LIN {X 0,Y 456.406,Z 1058.133,A -85,B 0,C 180,E1 19306.793,E2 19306.793} C_VEL
LIN {X 0,Y 463.105,Z 1034.289,A -85,B 0,C 180,E1 19306.028,E2 19306.028} C_VEL
LIN {X 0,Y 471.257,Z 1002.523,A -85,B 0,C 180,E1 19305.397,E2 19305.397} C_VEL
LIN {X 0,Y 477.978,Z 976.833,A -85,B 0,C 180,E1 19305.03,E2 19305.03} C_VEL
LIN {X 0,Y 462.437,Z 1036.182,A -85,B 0,C 180,E1 19303.259,E2 19303.259} C_VEL
LIN {X 0,Y 455.558,Z 1059.774,A -85,B 0,C 180,E1 19302.278,E2 19302.278} C_VEL
LIN {X 0,Y 447.956,Z 1083.299,A -85,B 0,C 180,E1 19301.014,E2 19301.014} C_VEL
LIN {X 0,Y 440.173,Z 1105.866,A -85,B 0,C 180,E1 19299.498,E2 19299.498} C_VEL
LIN {X 0,Y 432.109,Z 1128.201,A -85,B 0,C 180,E1 19297.654,E2 19297.654} C_VEL
LIN {X 0,Y 424.459,Z 1148.843,A -85,B 0,C 180,E1 19295.581,E2 19295.581} C_VEL
LIN {X 0,Y 417.628,Z 1166.966,A -85,B 0,C 180,E1 19293.413,E2 19293.413} C_VEL
LIN {X 0,Y 410.886,Z 1184.567,A -85,B 0,C 180,E1 19290.895,E2 19290.895} C_VEL
LIN {X 0,Y 404.741,Z 1200.504,A -85,B 0,C 180,E1 19288.155,E2 19288.155} C_VEL
LIN {X 0,Y 399.298,Z 1214.717,A -85,B 0,C 180,E1 19285.195,E2 19285.195} C_VEL
LIN {X 0,Y 395.001,Z 1226.059,A -85,B 0,C 180,E1 19282.315,E2 19282.315} C_VEL
LIN {X 0,Y 391.557,Z 1235.554,A -85,B 0,C 180,E1 19279.389,E2 19279.389} C_VEL
LIN {X 0,Y 388.794,Z 1243.686,A -85,B 0,C 180,E1 19276.28,E2 19276.28} C_VEL
LIN {X 0,Y 386.823,Z 1250.051,A -85,B 0,C 180,E1 19273.148,E2 19273.148} C_VEL
LIN {X 0,Y 385.498,Z 1254.602,A -85,B 0,C 180,E1 19270.008,E2 19270.008} C_VEL
LIN {X 0,Y 384.741,Z 1257.556,A -85,B 0,C 180,E1 19266.866,E2 19266.866} C_VEL
LIN {X 0,Y 384.358,Z 1258.935,A -85,B 0,C 180,E1 19263.878,E2 19263.878} C_VEL
LIN {X 0,Y 384.196,Z 1258.702,A -85,B 0,C 180,E1 19260.895,E2 19260.895} C_VEL
LIN {X 0,Y 384.141,Z 1256.912,A -85,B 0,C 180,E1 19257.762,E2 19257.762} C_VEL
LIN {X 0,Y 384.207,Z 1253.678,A -85,B 0,C 180,E1 19254.774,E2 19254.774} C_VEL
LIN {X 0,Y 384.45,Z 1248.721,A -85,B 0,C 180,E1 19251.776,E2 19251.776} C_VEL
LIN {X 0,Y 385.024,Z 1241.729,A -85,B 0,C 180,E1 19248.617,E2 19248.617} C_VEL
LIN {X 0,Y 385.962,Z 1233.447,A -85,B 0,C 180,E1 19245.678,E2 19245.678} C_VEL
LIN {X 0,Y 387.402,Z 1223.201,A -85,B 0,C 180,E1 19242.733,E2 19242.733} C_VEL
LIN {X 0,Y 389.23,Z 1211.755,A -85,B 0,C 180,E1 19240.022,E2 19240.022} C_VEL
LIN {X 0,Y 391.588,Z 1198.234,A -85,B 0,C 180,E1 19237.321,E2 19237.321} C_VEL
LIN {X 0,Y 394.348,Z 1183.215,A -85,B 0,C 180,E1 19234.788,E2 19234.788} C_VEL
LIN {X 0,Y 397.336,Z 1167.26,A -85,B 0,C 180,E1 19232.498,E2 19232.498} C_VEL
LIN {X 0,Y 400.703,Z 1148.832,A -85,B 0,C 180,E1 19230.273,E2 19230.273} C_VEL
LIN {X 0,Y 404.024,Z 1129.942,A -85,B 0,C 180,E1 19228.354,E2 19228.354} C_VEL
LIN {X 0,Y 407.3,Z 1109.911,A -85,B 0,C 180,E1 19226.639,E2 19226.639} C_VEL
LIN {X 0,Y 410.601,Z 1088.057,A -85,B 0,C 180,E1 19225.091,E2 19225.091} C_VEL
LIN {X 0,Y 413.484,Z 1066.4,A -85,B 0,C 180,E1 19223.84,E2 19223.84} C_VEL
LIN {X 0,Y 416.065,Z 1043.427,A -85,B 0,C 180,E1 19222.783,E2 19222.783} C_VEL
LIN {X 0,Y 418.284,Z 1019.214,A -85,B 0,C 180,E1 19221.949,E2 19221.949} C_VEL
LIN {X 0,Y 420.646,Z 982.191,A -85,B 0,C 180,E1 19221.071,E2 19221.071} C_VEL
LIN {X 0,Y 434.104,Z 779.214,A -85,B 0,C 180,E1 19216.578,E2 19216.578} C_VEL
LIN {X 0,Y 417.769,Z 747.187,A -85,B 0,C 180,E1 19214.052,E2 19214.052} C_VEL
LIN {X 0,Y 402.103,Z 718.746,A -85,B 0,C 180,E1 19211.46,E2 19211.46} C_VEL
LIN {X 0,Y 397.559,Z 710.697,A -85,B 0,C 180,E1 19210.649,E2 19210.649} C_VEL
LIN {X 0,Y 389.693,Z 691.665,A -85,B 0,C 180,E1 19207.269,E2 19207.269} C_VEL
LIN {X 0,Y 386.803,Z 684.581,A -85,B 0,C 180,E1 19205.973,E2 19205.973} C_VEL
LIN {X 0,Y 386.779,Z 684.484,A -85,B 0,C 180,E1 19201.83,E2 19201.83} C_VEL
LIN {X 0,Y 386.786,Z 684.485,A -85,B 0,C 180,E1 19197.857,E2 19197.857} C_VEL
LIN {X 0,Y 386.792,Z 684.486,A -85,B 0,C 180,E1 19193.776,E2 19193.776} C_VEL
LIN {X 0,Y 386.789,Z 684.485,A -85,B 0,C 180,E1 19189.783,E2 19189.783} C_VEL
LIN {X 0,Y 386.784,Z 684.488,A -85,B 0,C 180,E1 19185.752,E2 19185.752} C_VEL
LIN {X 0,Y 386.779,Z 684.483,A -85,B 0,C 180,E1 19181.786,E2 19181.786} C_VEL
LIN {X 0,Y 386.794,Z 684.472,A -85,B 0,C 180,E1 19177.727,E2 19177.727} C_VEL
LIN {X 0,Y 386.778,Z 684.475,A -85,B 0,C 180,E1 19173.708,E2 19173.708} C_VEL
LIN {X 0,Y 386.78,Z 684.474,A -85,B 0,C 180,E1 19169.706,E2 19169.706} C_VEL
LIN {X 0,Y 386.785,Z 684.475,A -85,B 0,C 180,E1 19165.703,E2 19165.703} C_VEL
LIN {X 0,Y 386.786,Z 684.478,A -85,B 0,C 180,E1 19161.678,E2 19161.678} C_VEL
LIN {X 0,Y 386.788,Z 684.487,A -85,B 0,C 180,E1 19157.612,E2 19157.612} C_VEL
LIN {X 0,Y 386.781,Z 684.489,A -85,B 0,C 180,E1 19153.636,E2 19153.636} C_VEL
LIN {X 0,Y 386.781,Z 684.483,A -85,B 0,C 180,E1 19149.577,E2 19149.577} C_VEL
LIN {X 0,Y 386.797,Z 684.617,A -85,B 0,C 180,E1 19146.592,E2 19146.592} C_VEL
LIN {X 0,Y 388.136,Z 688.034,A -85,B 0,C 180,E1 19145.823,E2 19145.823} C_VEL
LIN {X 0,Y 392.774,Z 697.922,A -85,B 0,C 180,E1 19143.547,E2 19143.547} C_VEL
LIN {X 0,Y 399.276,Z 712.504,A -85,B 0,C 180,E1 19140.443,E2 19140.443} C_VEL
LIN {X 0,Y 406.573,Z 730.369,A -85,B 0,C 180,E1 19136.996,E2 19136.996} C_VEL
LIN {X 0,Y 413.648,Z 749.213,A -85,B 0,C 180,E1 19133.688,E2 19133.688} C_VEL
LIN {X 0,Y 420.237,Z 768.718,A -85,B 0,C 180,E1 19130.562,E2 19130.562} C_VEL
LIN {X 0,Y 423.081,Z 778.482,A -85,B 0,C 180,E1 19129.11,E2 19129.11} C_VEL
LIN {X 0,Y 422.399,Z 782.605,A -85,B 0,C 180,E1 19128.699,E2 19128.699} C_VEL
LIN {X 0,Y 420.547,Z 788.964,A -85,B 0,C 180,E1 19128.148,E2 19128.148} C_VEL
LIN {X 0,Y 412.54,Z 806.493,A -85,B 0,C 180,E1 19126.91,E2 19126.91} C_VEL
LIN {X 0,Y 411.039,Z 811.959,A -85,B 0,C 180,E1 19126.42,E2 19126.42} C_VEL
LIN {X 0,Y 404.701,Z 854.209,A -85,B 0,C 180,E1 19122.17,E2 19122.17} C_VEL
LIN {X 0,Y 398.898,Z 897.769,A -85,B 0,C 180,E1 19117.807,E2 19117.807} C_VEL
LIN {X 0,Y 396.431,Z 919.14,A -85,B 0,C 180,E1 19115.714,E2 19115.714} C_VEL
LIN {X 0,Y 396.961,Z 931.506,A -85,B 0,C 180,E1 19115.277,E2 19115.277} C_VEL
LIN {X 0,Y 391.461,Z 1014.878,A -85,B 0,C 180,E1 19112.751,E2 19112.751} C_VEL
LIN {X 0,Y 388.582,Z 1066.505,A -85,B 0,C 180,E1 19110.979,E2 19110.979} C_VEL
LIN {X 0,Y 387.682,Z 1083.198,A -85,B 0,C 180,E1 19110.195,E2 19110.195} C_VEL
LIN {X 0,Y 386.441,Z 1100.03,A -85,B 0,C 180,E1 19109.107,E2 19109.107} C_VEL
LIN {X 0,Y 385.089,Z 1114.976,A -85,B 0,C 180,E1 19107.864,E2 19107.864} C_VEL
LIN {X 0,Y 383.556,Z 1130.549,A -85,B 0,C 180,E1 19106.233,E2 19106.233} C_VEL
LIN {X 0,Y 382.067,Z 1144.335,A -85,B 0,C 180,E1 19104.425,E2 19104.425} C_VEL
LIN {X 0,Y 380.789,Z 1156.067,A -85,B 0,C 180,E1 19102.543,E2 19102.543} C_VEL
LIN {X 0,Y 379.604,Z 1167.141,A -85,B 0,C 180,E1 19100.337,E2 19100.337} C_VEL
LIN {X 0,Y 378.783,Z 1175.987,A -85,B 0,C 180,E1 19098.148,E2 19098.148} C_VEL
LIN {X 0,Y 378.201,Z 1183.855,A -85,B 0,C 180,E1 19095.645,E2 19095.645} C_VEL
LIN {X 0,Y 377.967,Z 1189.648,A -85,B 0,C 180,E1 19093.15,E2 19093.15} C_VEL
LIN {X 0,Y 378.054,Z 1193.837,A -85,B 0,C 180,E1 19090.515,E2 19090.515} C_VEL
LIN {X 0,Y 378.485,Z 1196.093,A -85,B 0,C 180,E1 19087.896,E2 19087.896} C_VEL
LIN {X 0,Y 379.317,Z 1196.583,A -85,B 0,C 180,E1 19085.294,E2 19085.294} C_VEL
LIN {X 0,Y 380.693,Z 1195.118,A -85,B 0,C 180,E1 19082.559,E2 19082.559} C_VEL
LIN {X 0,Y 382.547,Z 1191.944,A -85,B 0,C 180,E1 19080,E2 19080} C_VEL
LIN {X 0,Y 384.988,Z 1186.906,A -85,B 0,C 180,E1 19077.469,E2 19077.469} C_VEL
LIN {X 0,Y 387.861,Z 1180.364,A -85,B 0,C 180,E1 19075.12,E2 19075.12} C_VEL
LIN {X 0,Y 391.295,Z 1171.875,A -85,B 0,C 180,E1 19072.807,E2 19072.807} C_VEL
LIN {X 0,Y 395.366,Z 1160.869,A -85,B 0,C 180,E1 19070.494,E2 19070.494} C_VEL
LIN {X 0,Y 399.536,Z 1148.444,A -85,B 0,C 180,E1 19068.451,E2 19068.451} C_VEL
LIN {X 0,Y 403.782,Z 1134.322,A -85,B 0,C 180,E1 19066.612,E2 19066.612} C_VEL
LIN {X 0,Y 407.497,Z 1120.527,A -85,B 0,C 180,E1 19065.178,E2 19065.178} C_VEL
LIN {X 0,Y 411.082,Z 1105.238,A -85,B 0,C 180,E1 19063.902,E2 19063.902} C_VEL
LIN {X 0,Y 414.429,Z 1088.699,A -85,B 0,C 180,E1 19062.809,E2 19062.809} C_VEL
LIN {X 0,Y 421.189,Z 1056.224,A -85,B 0,C 180,E1 19061.092,E2 19061.092} C_VEL
LIN {X 0,Y 430.656,Z 1013.251,A -85,B 0,C 180,E1 19059.228,E2 19059.228} C_VEL
LIN {X 0,Y 438.334,Z 973.633,A -85,B 0,C 180,E1 19057.784,E2 19057.784} C_VEL
LIN {X 0,Y 441.205,Z 956.554,A -85,B 0,C 180,E1 19057.208,E2 19057.208} C_VEL
LIN {X 0,Y 441.342,Z 949.51,A -85,B 0,C 180,E1 19056.642,E2 19056.642} C_VEL
LIN {X 0,Y 454.238,Z 919.763,A -85,B 0,C 180,E1 19053.034,E2 19053.034} C_VEL
LIN {X 0,Y 469.215,Z 891.646,A -85,B 0,C 180,E1 19049.524,E2 19049.524} C_VEL
LIN {X 0,Y 481.049,Z 873.153,A -85,B 0,C 180,E1 19047.145,E2 19047.145} C_VEL
LIN {X 0,Y 469,Z 892.326,A -85,B 0,C 180,E1 19044.856,E2 19044.856} C_VEL
LIN {X 0,Y 459.771,Z 910.769,A -85,B 0,C 180,E1 19042.434,E2 19042.434} C_VEL
LIN {X 0,Y 453.792,Z 927.463,A -85,B 0,C 180,E1 19040.062,E2 19040.062} C_VEL
LIN {X 0,Y 450.252,Z 944.409,A -85,B 0,C 180,E1 19037.497,E2 19037.497} C_VEL
LIN {X 0,Y 449.463,Z 960.306,A -85,B 0,C 180,E1 19034.973,E2 19034.973} C_VEL
LIN {X 0,Y 449.631,Z 965.006,A -85,B 0,C 180,E1 19034.241,E2 19034.241} C_VEL
LIN {X 0,Y 440.372,Z 984.021,A -85,B 0,C 180,E1 19033.366,E2 19033.366} C_VEL
LIN {X 0,Y 437.358,Z 1002.491,A -85,B 0,C 180,E1 19033.036,E2 19033.036} C_VEL
LIN {X 0,Y 432.995,Z 1027.628,A -85,B 0,C 180,E1 19032.57,E2 19032.57} C_VEL
LIN {X 0,Y 428.798,Z 1050.895,A -85,B 0,C 180,E1 19031.825,E2 19031.825} C_VEL
LIN {X 0,Y 423.742,Z 1075.158,A -85,B 0,C 180,E1 19030.812,E2 19030.812} C_VEL
LIN {X 0,Y 418.025,Z 1099.477,A -85,B 0,C 180,E1 19029.51,E2 19029.51} C_VEL
LIN {X 0,Y 412.366,Z 1121.842,A -85,B 0,C 180,E1 19028.013,E2 19028.013} C_VEL
LIN {X 0,Y 406.51,Z 1143.789,A -85,B 0,C 180,E1 19026.217,E2 19026.217} C_VEL
LIN {X 0,Y 400.803,Z 1164.727,A -85,B 0,C 180,E1 19024.143,E2 19024.143} C_VEL
LIN {X 0,Y 395.713,Z 1183.09,A -85,B 0,C 180,E1 19021.96,E2 19021.96} C_VEL
LIN {X 0,Y 390.742,Z 1201.05,A -85,B 0,C 180,E1 19019.424,E2 19019.424} C_VEL
LIN {X 0,Y 386.333,Z 1217.744,A -85,B 0,C 180,E1 19016.597,E2 19016.597} C_VEL
LIN {X 0,Y 382.67,Z 1232.679,A -85,B 0,C 180,E1 19013.562,E2 19013.562} C_VEL
LIN {X 0,Y 380.6,Z 1242.938,A -85,B 0,C 180,E1 19011.254,E2 19011.254} C_VEL
LIN {X 0,Y 378.702,Z 1255.869,A -85,B 0,C 180,E1 19008.31,E2 19008.31} C_VEL
LIN {X 0,Y 377.462,Z 1266.125,A -85,B 0,C 180,E1 19005.516,E2 19005.516} C_VEL
LIN {X 0,Y 376.686,Z 1274.965,A -85,B 0,C 180,E1 19002.57,E2 19002.57} C_VEL
LIN {X 0,Y 376.336,Z 1281.925,A -85,B 0,C 180,E1 18999.634,E2 18999.634} C_VEL
LIN {X 0,Y 376.272,Z 1287.256,A -85,B 0,C 180,E1 18996.712,E2 18996.712} C_VEL
LIN {X 0,Y 376.329,Z 1290.731,A -85,B 0,C 180,E1 18993.959,E2 18993.959} C_VEL
LIN {X 0,Y 376.375,Z 1292.953,A -85,B 0,C 180,E1 18991.063,E2 18991.063} C_VEL
LIN {X 0,Y 376.318,Z 1293.599,A -85,B 0,C 180,E1 18988.323,E2 18988.323} C_VEL
LIN {X 0,Y 376.183,Z 1292.797,A -85,B 0,C 180,E1 18985.272,E2 18985.272} C_VEL
LIN {X 0,Y 376.148,Z 1290.524,A -85,B 0,C 180,E1 18982.36,E2 18982.36} C_VEL
LIN {X 0,Y 376.396,Z 1286.334,A -85,B 0,C 180,E1 18979.126,E2 18979.126} C_VEL
LIN {X 0,Y 377.218,Z 1280.438,A -85,B 0,C 180,E1 18975.883,E2 18975.883} C_VEL
LIN {X 0,Y 378.757,Z 1272.659,A -85,B 0,C 180,E1 18972.642,E2 18972.642} C_VEL
LIN {X 0,Y 381.096,Z 1263.219,A -85,B 0,C 180,E1 18969.5,E2 18969.5} C_VEL
LIN {X 0,Y 384.396,Z 1251.872,A -85,B 0,C 180,E1 18966.383,E2 18966.383} C_VEL
LIN {X 0,Y 388.594,Z 1238.846,A -85,B 0,C 180,E1 18963.401,E2 18963.401} C_VEL
LIN {X 0,Y 393.824,Z 1223.589,A -85,B 0,C 180,E1 18960.49,E2 18960.49} C_VEL
LIN {X 0,Y 399.81,Z 1206.907,A -85,B 0,C 180,E1 18957.811,E2 18957.811} C_VEL
LIN {X 0,Y 406.875,Z 1187.889,A -85,B 0,C 180,E1 18955.239,E2 18955.239} C_VEL
LIN {X 0,Y 414.857,Z 1166.814,A -85,B 0,C 180,E1 18952.859,E2 18952.859} C_VEL
LIN {X 0,Y 423.268,Z 1144.944,A -85,B 0,C 180,E1 18950.807,E2 18950.807} C_VEL
LIN {X 0,Y 432.218,Z 1121.656,A -85,B 0,C 180,E1 18949.015,E2 18949.015} C_VEL
LIN {X 0,Y 441.303,Z 1097.605,A -85,B 0,C 180,E1 18947.529,E2 18947.529} C_VEL
LIN {X 0,Y 449.996,Z 1073.504,A -85,B 0,C 180,E1 18946.374,E2 18946.374} C_VEL
LIN {X 0,Y 458.572,Z 1047.367,A -85,B 0,C 180,E1 18945.403,E2 18945.403} C_VEL
LIN {X 0,Y 464.318,Z 1027.702,A -85,B 0,C 180,E1 18944.876,E2 18944.876} C_VEL
LIN {X 0,Y 465.978,Z 1021.566,A -85,B 0,C 180,E1 18944.745,E2 18944.745} C_VEL
LIN {X 0,Y 459.374,Z 1044.375,A -85,B 0,C 180,E1 18943.976,E2 18943.976} C_VEL
LIN {X 0,Y 451.876,Z 1067.125,A -85,B 0,C 180,E1 18942.963,E2 18942.963} C_VEL
LIN {X 0,Y 443.67,Z 1089.81,A -85,B 0,C 180,E1 18941.67,E2 18941.67} C_VEL
LIN {X 0,Y 435.273,Z 1111.647,A -85,B 0,C 180,E1 18940.117,E2 18940.117} C_VEL
LIN {X 0,Y 426.625,Z 1133.377,A -85,B 0,C 180,E1 18938.225,E2 18938.225} C_VEL
LIN {X 0,Y 418.205,Z 1154.079,A -85,B 0,C 180,E1 18936.027,E2 18936.027} C_VEL
LIN {X 0,Y 410.704,Z 1172.232,A -85,B 0,C 180,E1 18933.717,E2 18933.717} C_VEL
LIN {X 0,Y 403.747,Z 1188.938,A -85,B 0,C 180,E1 18931.171,E2 18931.171} C_VEL
LIN {X 0,Y 397.39,Z 1204.141,A -85,B 0,C 180,E1 18928.395,E2 18928.395} C_VEL
LIN {X 0,Y 392.009,Z 1217.156,A -85,B 0,C 180,E1 18925.535,E2 18925.535} C_VEL
LIN {X 0,Y 387.542,Z 1228.201,A -85,B 0,C 180,E1 18922.609,E2 18922.609} C_VEL
LIN {X 0,Y 383.621,Z 1238.188,A -85,B 0,C 180,E1 18919.331,E2 18919.331} C_VEL
LIN {X 0,Y 380.794,Z 1245.781,A -85,B 0,C 180,E1 18916.161,E2 18916.161} C_VEL
LIN {X 0,Y 378.709,Z 1251.902,A -85,B 0,C 180,E1 18912.814,E2 18912.814} C_VEL
LIN {X 0,Y 377.424,Z 1256.07,A -85,B 0,C 180,E1 18909.608,E2 18909.608} C_VEL
LIN {X 0,Y 376.69,Z 1258.572,A -85,B 0,C 180,E1 18906.401,E2 18906.401} C_VEL
LIN {X 0,Y 376.324,Z 1259.428,A -85,B 0,C 180,E1 18903.351,E2 18903.351} C_VEL
LIN {X 0,Y 376.185,Z 1258.887,A -85,B 0,C 180,E1 18900.305,E2 18900.305} C_VEL
LIN {X 0,Y 376.145,Z 1256.734,A -85,B 0,C 180,E1 18897.257,E2 18897.257} C_VEL
LIN {X 0,Y 376.249,Z 1252.844,A -85,B 0,C 180,E1 18894.051,E2 18894.051} C_VEL
LIN {X 0,Y 376.567,Z 1247.507,A -85,B 0,C 180,E1 18890.987,E2 18890.987} C_VEL
LIN {X 0,Y 377.207,Z 1240.368,A -85,B 0,C 180,E1 18887.912,E2 18887.912} C_VEL
LIN {X 0,Y 378.241,Z 1231.8,A -85,B 0,C 180,E1 18884.985,E2 18884.985} C_VEL
LIN {X 0,Y 379.78,Z 1221.393,A -85,B 0,C 180,E1 18882.059,E2 18882.059} C_VEL
LIN {X 0,Y 381.841,Z 1209.2,A -85,B 0,C 180,E1 18879.206,E2 18879.206} C_VEL
LIN {X 0,Y 384.305,Z 1195.565,A -85,B 0,C 180,E1 18876.542,E2 18876.542} C_VEL
LIN {X 0,Y 387.058,Z 1180.913,A -85,B 0,C 180,E1 18874.114,E2 18874.114} C_VEL
LIN {X 0,Y 390.418,Z 1163.27,A -85,B 0,C 180,E1 18871.635,E2 18871.635} C_VEL
LIN {X 0,Y 393.815,Z 1145.086,A -85,B 0,C 180,E1 18869.483,E2 18869.483} C_VEL
LIN {X 0,Y 397.221,Z 1126.038,A -85,B 0,C 180,E1 18867.577,E2 18867.577} C_VEL
LIN {X 0,Y 400.659,Z 1105.262,A -85,B 0,C 180,E1 18865.839,E2 18865.839} C_VEL
LIN {X 0,Y 403.876,Z 1083.883,A -85,B 0,C 180,E1 18864.371,E2 18864.371} C_VEL
LIN {X 0,Y 406.75,Z 1061.916,A -85,B 0,C 180,E1 18863.143,E2 18863.143} C_VEL
LIN {X 0,Y 409.362,Z 1038.294,A -85,B 0,C 180,E1 18862.104,E2 18862.104} C_VEL
LIN {X 0,Y 411.49,Z 1014.34,A -85,B 0,C 180,E1 18861.321,E2 18861.321} C_VEL
LIN {X 0,Y 427.32,Z 781.831,A -85,B 0,C 180,E1 18856.026,E2 18856.026} C_VEL
LIN {X 0,Y 411.74,Z 751.237,A -85,B 0,C 180,E1 18853.558,E2 18853.558} C_VEL
LIN {X 0,Y 396.564,Z 723.52,A -85,B 0,C 180,E1 18850.988,E2 18850.988} C_VEL
LIN {X 0,Y 389.539,Z 711.201,A -85,B 0,C 180,E1 18849.73,E2 18849.73} C_VEL
LIN {X 0,Y 382.044,Z 693.158,A -85,B 0,C 180,E1 18846.451,E2 18846.451} C_VEL
LIN {X 0,Y 378.868,Z 685.654,A -85,B 0,C 180,E1 18845.026,E2 18845.026} C_VEL
LIN {X 0,Y 378.858,Z 685.462,A -85,B 0,C 180,E1 18840.935,E2 18840.935} C_VEL
LIN {X 0,Y 378.845,Z 685.478,A -85,B 0,C 180,E1 18836.83,E2 18836.83} C_VEL
LIN {X 0,Y 378.852,Z 685.478,A -85,B 0,C 180,E1 18832.83,E2 18832.83} C_VEL
LIN {X 0,Y 378.85,Z 685.474,A -85,B 0,C 180,E1 18828.785,E2 18828.785} C_VEL
LIN {X 0,Y 378.853,Z 685.472,A -85,B 0,C 180,E1 18824.679,E2 18824.679} C_VEL
LIN {X 0,Y 378.849,Z 685.477,A -85,B 0,C 180,E1 18820.648,E2 18820.648} C_VEL
LIN {X 0,Y 378.843,Z 685.477,A -85,B 0,C 180,E1 18816.519,E2 18816.519} C_VEL
LIN {X 0,Y 378.841,Z 685.476,A -85,B 0,C 180,E1 18812.422,E2 18812.422} C_VEL
LIN {X 0,Y 378.854,Z 685.472,A -85,B 0,C 180,E1 18808.49,E2 18808.49} C_VEL
LIN {X 0,Y 378.841,Z 685.479,A -85,B 0,C 180,E1 18804.29,E2 18804.29} C_VEL
LIN {X 0,Y 378.842,Z 685.477,A -85,B 0,C 180,E1 18800.124,E2 18800.124} C_VEL
LIN {X 0,Y 378.854,Z 685.469,A -85,B 0,C 180,E1 18796.106,E2 18796.106} C_VEL
LIN {X 0,Y 378.844,Z 685.474,A -85,B 0,C 180,E1 18792.016,E2 18792.016} C_VEL
LIN {X 0,Y 378.862,Z 685.613,A -85,B 0,C 180,E1 18787.875,E2 18787.875} C_VEL
LIN {X 0,Y 380.166,Z 688.967,A -85,B 0,C 180,E1 18787.094,E2 18787.094} C_VEL
LIN {X 0,Y 381.28,Z 691.358,A -85,B 0,C 180,E1 18786.511,E2 18786.511} C_VEL
LIN {X 0,Y 385.024,Z 699.228,A -85,B 0,C 180,E1 18784.63,E2 18784.63} C_VEL
LIN {X 0,Y 391.461,Z 713.489,A -85,B 0,C 180,E1 18781.471,E2 18781.471} C_VEL
LIN {X 0,Y 398.706,Z 731.085,A -85,B 0,C 180,E1 18777.957,E2 18777.957} C_VEL
LIN {X 0,Y 405.713,Z 749.515,A -85,B 0,C 180,E1 18774.611,E2 18774.611} C_VEL
LIN {X 0,Y 412.248,Z 768.67,A -85,B 0,C 180,E1 18771.443,E2 18771.443} C_VEL
LIN {X 0,Y 416.081,Z 780.955,A -85,B 0,C 180,E1 18769.549,E2 18769.549} C_VEL
LIN {X 0,Y 411.039,Z 811.959,A -85,B 0,C 180,E1 18766.42,E2 18766.42} C_VEL
LIN {X 0,Y 409.194,Z 818.344,A -85,B 0,C 180,E1 18765.857,E2 18765.857} C_VEL
LIN {X 0,Y 401.155,Z 835.87,A -85,B 0,C 180,E1 18764.586,E2 18764.586} C_VEL
LIN {X 0,Y 399.672,Z 841.352,A -85,B 0,C 180,E1 18764.087,E2 18764.087} C_VEL
LIN {X 0,Y 393.527,Z 883.988,A -85,B 0,C 180,E1 18759.754,E2 18759.754} C_VEL
LIN {X 0,Y 389.047,Z 919.915,A -85,B 0,C 180,E1 18756.153,E2 18756.153} C_VEL
LIN {X 0,Y 389.547,Z 932.135,A -85,B 0,C 180,E1 18755.712,E2 18755.712} C_VEL
LIN {X 0,Y 384.099,Z 1012.065,A -85,B 0,C 180,E1 18753.236,E2 18753.236} C_VEL
LIN {X 0,Y 380.975,Z 1064.895,A -85,B 0,C 180,E1 18751.377,E2 18751.377} C_VEL
LIN {X 0,Y 379.978,Z 1083.049,A -85,B 0,C 180,E1 18750.522,E2 18750.522} C_VEL
LIN {X 0,Y 378.672,Z 1100.387,A -85,B 0,C 180,E1 18749.388,E2 18749.388} C_VEL
LIN {X 0,Y 377.311,Z 1115.165,A -85,B 0,C 180,E1 18748.145,E2 18748.145} C_VEL
LIN {X 0,Y 375.723,Z 1130.908,A -85,B 0,C 180,E1 18746.472,E2 18746.472} C_VEL
LIN {X 0,Y 374.273,Z 1144.099,A -85,B 0,C 180,E1 18744.732,E2 18744.732} C_VEL
LIN {X 0,Y 372.885,Z 1156.564,A -85,B 0,C 180,E1 18742.714,E2 18742.714} C_VEL
LIN {X 0,Y 371.738,Z 1167.073,A -85,B 0,C 180,E1 18740.612,E2 18740.612} C_VEL
LIN {X 0,Y 370.825,Z 1176.644,A -85,B 0,C 180,E1 18738.227,E2 18738.227} C_VEL
LIN {X 0,Y 370.228,Z 1184.56,A -85,B 0,C 180,E1 18735.669,E2 18735.669} C_VEL
LIN {X 0,Y 370,Z 1190.47,A -85,B 0,C 180,E1 18733.121,E2 18733.121} C_VEL
LIN {X 0,Y 370.104,Z 1194.741,A -85,B 0,C 180,E1 18730.429,E2 18730.429} C_VEL
LIN {X 0,Y 370.536,Z 1197.031,A -85,B 0,C 180,E1 18727.91,E2 18727.91} C_VEL
LIN {X 0,Y 371.465,Z 1197.7,A -85,B 0,C 180,E1 18725.096,E2 18725.096} C_VEL
LIN {X 0,Y 372.834,Z 1196.485,A -85,B 0,C 180,E1 18722.459,E2 18722.459} C_VEL
LIN {X 0,Y 374.77,Z 1193.56,A -85,B 0,C 180,E1 18719.847,E2 18719.847} C_VEL
LIN {X 0,Y 377.484,Z 1188.452,A -85,B 0,C 180,E1 18717.115,E2 18717.115} C_VEL
LIN {X 0,Y 380.508,Z 1182.076,A -85,B 0,C 180,E1 18714.723,E2 18714.723} C_VEL
LIN {X 0,Y 384.357,Z 1173.217,A -85,B 0,C 180,E1 18712.225,E2 18712.225} C_VEL
LIN {X 0,Y 388.581,Z 1162.578,A -85,B 0,C 180,E1 18709.923,E2 18709.923} C_VEL
LIN {X 0,Y 393.057,Z 1150.086,A -85,B 0,C 180,E1 18707.811,E2 18707.811} C_VEL
LIN {X 0,Y 397.184,Z 1137.362,A -85,B 0,C 180,E1 18706.089,E2 18706.089} C_VEL
LIN {X 0,Y 401.334,Z 1123.096,A -85,B 0,C 180,E1 18704.539,E2 18704.539} C_VEL
LIN {X 0,Y 405.231,Z 1108.051,A -85,B 0,C 180,E1 18703.22,E2 18703.22} C_VEL
LIN {X 0,Y 408.927,Z 1091.019,A -85,B 0,C 180,E1 18702.056,E2 18702.056} C_VEL
LIN {X 0,Y 415.659,Z 1060.815,A -85,B 0,C 180,E1 18700.392,E2 18700.392} C_VEL
LIN {X 0,Y 424.645,Z 1022.682,A -85,B 0,C 180,E1 18698.667,E2 18698.667} C_VEL
LIN {X 0,Y 432.253,Z 986.723,A -85,B 0,C 180,E1 18697.284,E2 18697.284} C_VEL
LIN {X 0,Y 437.347,Z 958.876,A -85,B 0,C 180,E1 18696.326,E2 18696.326} C_VEL
LIN {X 0,Y 437.68,Z 950.75,A -85,B 0,C 180,E1 18695.647,E2 18695.647} C_VEL
LIN {X 0,Y 452.407,Z 919.337,A -85,B 0,C 180,E1 18691.772,E2 18691.772} C_VEL
LIN {X 0,Y 467.712,Z 892.826,A -85,B 0,C 180,E1 18688.414,E2 18688.414} C_VEL
LIN {X 0,Y 473.959,Z 883.438,A -85,B 0,C 180,E1 18687.181,E2 18687.181} C_VEL
LIN {X 0,Y 462.006,Z 902.676,A -85,B 0,C 180,E1 18684.781,E2 18684.781} C_VEL
LIN {X 0,Y 453.164,Z 920.878,A -85,B 0,C 180,E1 18682.287,E2 18682.287} C_VEL
LIN {X 0,Y 447.676,Z 936.946,A -85,B 0,C 180,E1 18679.901,E2 18679.901} C_VEL
LIN {X 0,Y 444.488,Z 954.093,A -85,B 0,C 180,E1 18677.206,E2 18677.206} C_VEL
LIN {X 0,Y 443.966,Z 967.723,A -85,B 0,C 180,E1 18674.993,E2 18674.993} C_VEL
LIN {X 0,Y 436.582,Z 982.675,A -85,B 0,C 180,E1 18674.306,E2 18674.306} C_VEL
LIN {X 0,Y 433.672,Z 1000.523,A -85,B 0,C 180,E1 18673.972,E2 18673.972} C_VEL
LIN {X 0,Y 428.845,Z 1026.946,A -85,B 0,C 180,E1 18673.489,E2 18673.489} C_VEL
LIN {X 0,Y 424.777,Z 1048.231,A -85,B 0,C 180,E1 18672.816,E2 18672.816} C_VEL
LIN {X 0,Y 419.077,Z 1074.204,A -85,B 0,C 180,E1 18671.731,E2 18671.731} C_VEL
LIN {X 0,Y 413.108,Z 1098.249,A -85,B 0,C 180,E1 18670.438,E2 18670.438} C_VEL
LIN {X 0,Y 406.955,Z 1121.298,A -85,B 0,C 180,E1 18668.882,E2 18668.882} C_VEL
LIN {X 0,Y 400.709,Z 1143.313,A -85,B 0,C 180,E1 18667.054,E2 18667.054} C_VEL
LIN {X 0,Y 394.978,Z 1163.142,A -85,B 0,C 180,E1 18665.072,E2 18665.072} C_VEL
LIN {X 0,Y 389.394,Z 1182.01,A -85,B 0,C 180,E1 18662.804,E2 18662.804} C_VEL
LIN {X 0,Y 384.246,Z 1199.367,A -85,B 0,C 180,E1 18660.317,E2 18660.317} C_VEL
LIN {X 0,Y 379.72,Z 1215.297,A -85,B 0,C 180,E1 18657.607,E2 18657.607} C_VEL
LIN {X 0,Y 375.679,Z 1230.398,A -85,B 0,C 180,E1 18654.529,E2 18654.529} C_VEL
LIN {X 0,Y 371.87,Z 1247.819,A -85,B 0,C 180,E1 18650.293,E2 18650.293} C_VEL
LIN {X 0,Y 370.244,Z 1259.363,A -85,B 0,C 180,E1 18647.441,E2 18647.441} C_VEL
LIN {X 0,Y 369.115,Z 1269.385,A -85,B 0,C 180,E1 18644.429,E2 18644.429} C_VEL
LIN {X 0,Y 368.509,Z 1277.464,A -85,B 0,C 180,E1 18641.422,E2 18641.422} C_VEL
LIN {X 0,Y 368.301,Z 1283.828,A -85,B 0,C 180,E1 18638.428,E2 18638.428} C_VEL
LIN {X 0,Y 368.311,Z 1288.235,A -85,B 0,C 180,E1 18635.606,E2 18635.606} C_VEL
LIN {X 0,Y 368.38,Z 1291.479,A -85,B 0,C 180,E1 18632.487,E2 18632.487} C_VEL
LIN {X 0,Y 368.373,Z 1292.944,A -85,B 0,C 180,E1 18629.687,E2 18629.687} C_VEL
LIN {X 0,Y 368.248,Z 1292.955,A -85,B 0,C 180,E1 18626.573,E2 18626.573} C_VEL
LIN {X 0,Y 368.137,Z 1291.514,A -85,B 0,C 180,E1 18623.604,E2 18623.604} C_VEL
LIN {X 0,Y 368.239,Z 1288.362,A -85,B 0,C 180,E1 18620.464,E2 18620.464} C_VEL
LIN {X 0,Y 368.823,Z 1283.437,A -85,B 0,C 180,E1 18617.154,E2 18617.154} C_VEL
LIN {X 0,Y 370.092,Z 1276.707,A -85,B 0,C 180,E1 18613.841,E2 18613.841} C_VEL
LIN {X 0,Y 372.231,Z 1268.097,A -85,B 0,C 180,E1 18610.538,E2 18610.538} C_VEL
LIN {X 0,Y 375.529,Z 1257.049,A -85,B 0,C 180,E1 18607.113,E2 18607.113} C_VEL
LIN {X 0,Y 379.775,Z 1244.489,A -85,B 0,C 180,E1 18603.914,E2 18603.914} C_VEL
LIN {X 0,Y 384.929,Z 1230.458,A -85,B 0,C 180,E1 18600.937,E2 18600.937} C_VEL
LIN {X 0,Y 391.164,Z 1214.188,A -85,B 0,C 180,E1 18598.051,E2 18598.051} C_VEL
LIN {X 0,Y 398.198,Z 1196.551,A -85,B 0,C 180,E1 18595.423,E2 18595.423} C_VEL
LIN {X 0,Y 406.384,Z 1176.641,A -85,B 0,C 180,E1 18592.927,E2 18592.927} C_VEL
LIN {X 0,Y 415.548,Z 1154.745,A -85,B 0,C 180,E1 18590.65,E2 18590.65} C_VEL
LIN {X 0,Y 425.126,Z 1132.072,A -85,B 0,C 180,E1 18588.719,E2 18588.719} C_VEL
LIN {X 0,Y 434.588,Z 1109.569,A -85,B 0,C 180,E1 18587.164,E2 18587.164} C_VEL
LIN {X 0,Y 443.643,Z 1087.359,A -85,B 0,C 180,E1 18585.947,E2 18585.947} C_VEL
LIN {X 0,Y 452.71,Z 1063.579,A -85,B 0,C 180,E1 18584.936,E2 18584.936} C_VEL
LIN {X 0,Y 455.839,Z 1054.673,A -85,B 0,C 180,E1 18584.604,E2 18584.604} C_VEL
LIN {X 0,Y 447.71,Z 1076.425,A -85,B 0,C 180,E1 18583.55,E2 18583.55} C_VEL
LIN {X 0,Y 438.917,Z 1098.063,A -85,B 0,C 180,E1 18582.225,E2 18582.225} C_VEL
LIN {X 0,Y 429.386,Z 1120.298,A -85,B 0,C 180,E1 18580.519,E2 18580.519} C_VEL
LIN {X 0,Y 420.24,Z 1141.063,A -85,B 0,C 180,E1 18578.564,E2 18578.564} C_VEL
LIN {X 0,Y 411.332,Z 1160.944,A -85,B 0,C 180,E1 18576.293,E2 18576.293} C_VEL
LIN {X 0,Y 403.249,Z 1178.853,A -85,B 0,C 180,E1 18573.831,E2 18573.831} C_VEL
LIN {X 0,Y 395.943,Z 1194.953,A -85,B 0,C 180,E1 18571.178,E2 18571.178} C_VEL
LIN {X 0,Y 389.49,Z 1209.229,A -85,B 0,C 180,E1 18568.355,E2 18568.355} C_VEL
LIN {X 0,Y 383.731,Z 1222.023,A -85,B 0,C 180,E1 18565.284,E2 18565.284} C_VEL
LIN {X 0,Y 379.05,Z 1232.643,A -85,B 0,C 180,E1 18562.162,E2 18562.162} C_VEL
LIN {X 0,Y 375.34,Z 1241.42,A -85,B 0,C 180,E1 18558.964,E2 18558.964} C_VEL
LIN {X 0,Y 372.556,Z 1248.446,A -85,B 0,C 180,E1 18555.728,E2 18555.728} C_VEL
LIN {X 0,Y 370.536,Z 1253.993,A -85,B 0,C 180,E1 18552.309,E2 18552.309} C_VEL
LIN {X 0,Y 369.251,Z 1257.652,A -85,B 0,C 180,E1 18548.879,E2 18548.879} C_VEL
LIN {X 0,Y 368.581,Z 1259.529,A -85,B 0,C 180,E1 18545.605,E2 18545.605} C_VEL
LIN {X 0,Y 368.279,Z 1259.893,A -85,B 0,C 180,E1 18542.49,E2 18542.49} C_VEL
LIN {X 0,Y 368.178,Z 1258.657,A -85,B 0,C 180,E1 18539.378,E2 18539.378} C_VEL
LIN {X 0,Y 368.161,Z 1255.776,A -85,B 0,C 180,E1 18536.107,E2 18536.107} C_VEL
LIN {X 0,Y 368.334,Z 1251.464,A -85,B 0,C 180,E1 18532.983,E2 18532.983} C_VEL
LIN {X 0,Y 368.723,Z 1245.71,A -85,B 0,C 180,E1 18530.005,E2 18530.005} C_VEL
LIN {X 0,Y 369.526,Z 1237.942,A -85,B 0,C 180,E1 18526.862,E2 18526.862} C_VEL
LIN {X 0,Y 370.747,Z 1228.781,A -85,B 0,C 180,E1 18523.872,E2 18523.872} C_VEL
LIN {X 0,Y 372.526,Z 1217.589,A -85,B 0,C 180,E1 18520.877,E2 18520.877} C_VEL
LIN {X 0,Y 374.758,Z 1204.949,A -85,B 0,C 180,E1 18518.066,E2 18518.066} C_VEL
LIN {X 0,Y 377.412,Z 1190.878,A -85,B 0,C 180,E1 18515.421,E2 18515.421} C_VEL
LIN {X 0,Y 380.528,Z 1174.908,A -85,B 0,C 180,E1 18512.877,E2 18512.877} C_VEL
LIN {X 0,Y 383.827,Z 1157.995,A -85,B 0,C 180,E1 18510.59,E2 18510.59} C_VEL
LIN {X 0,Y 387.447,Z 1138.78,A -85,B 0,C 180,E1 18508.407,E2 18508.407} C_VEL
LIN {X 0,Y 390.917,Z 1119.268,A -85,B 0,C 180,E1 18506.55,E2 18506.55} C_VEL
LIN {X 0,Y 394.249,Z 1099.078,A -85,B 0,C 180,E1 18504.939,E2 18504.939} C_VEL
LIN {X 0,Y 397.499,Z 1077.144,A -85,B 0,C 180,E1 18503.494,E2 18503.494} C_VEL
LIN {X 0,Y 400.343,Z 1055.214,A -85,B 0,C 180,E1 18502.327,E2 18502.327} C_VEL
LIN {X 0,Y 402.879,Z 1031.797,A -85,B 0,C 180,E1 18501.354,E2 18501.354} C_VEL
LIN {X 0,Y 404.925,Z 1007.074,A -85,B 0,C 180,E1 18500.608,E2 18500.608} C_VEL
LIN {X 0,Y 420.632,Z 784.541,A -85,B 0,C 180,E1 18495.468,E2 18495.468} C_VEL
LIN {X 0,Y 404.437,Z 752.762,A -85,B 0,C 180,E1 18492.836,E2 18492.836} C_VEL
LIN {X 0,Y 388.875,Z 724.49,A -85,B 0,C 180,E1 18490.124,E2 18490.124} C_VEL
LIN {X 0,Y 381.361,Z 711.348,A -85,B 0,C 180,E1 18488.708,E2 18488.708} C_VEL
LIN {X 0,Y 374.042,Z 693.994,A -85,B 0,C 180,E1 18485.458,E2 18485.458} C_VEL
LIN {X 0,Y 370.934,Z 686.681,A -85,B 0,C 180,E1 18484.038,E2 18484.038} C_VEL
LIN {X 0,Y 370.912,Z 686.455,A -85,B 0,C 180,E1 18480.078,E2 18480.078} C_VEL
LIN {X 0,Y 370.907,Z 686.464,A -85,B 0,C 180,E1 18476.068,E2 18476.068} C_VEL
LIN {X 0,Y 370.911,Z 686.465,A -85,B 0,C 180,E1 18471.975,E2 18471.975} C_VEL
LIN {X 0,Y 370.91,Z 686.466,A -85,B 0,C 180,E1 18467.896,E2 18467.896} C_VEL
LIN {X 0,Y 370.904,Z 686.452,A -85,B 0,C 180,E1 18463.725,E2 18463.725} C_VEL
LIN {X 0,Y 370.902,Z 686.458,A -85,B 0,C 180,E1 18459.624,E2 18459.624} C_VEL
LIN {X 0,Y 370.908,Z 686.464,A -85,B 0,C 180,E1 18455.571,E2 18455.571} C_VEL
LIN {X 0,Y 370.902,Z 686.467,A -85,B 0,C 180,E1 18451.392,E2 18451.392} C_VEL
LIN {X 0,Y 370.901,Z 686.464,A -85,B 0,C 180,E1 18447.221,E2 18447.221} C_VEL
LIN {X 0,Y 370.905,Z 686.46,A -85,B 0,C 180,E1 18443.19,E2 18443.19} C_VEL
LIN {X 0,Y 370.898,Z 686.456,A -85,B 0,C 180,E1 18439.125,E2 18439.125} C_VEL
LIN {X 0,Y 370.904,Z 686.46,A -85,B 0,C 180,E1 18435.004,E2 18435.004} C_VEL
LIN {X 0,Y 370.914,Z 686.467,A -85,B 0,C 180,E1 18430.965,E2 18430.965} C_VEL
LIN {X 0,Y 370.928,Z 686.612,A -85,B 0,C 180,E1 18429.227,E2 18429.227} C_VEL
LIN {X 0,Y 372.236,Z 689.985,A -85,B 0,C 180,E1 18428.41,E2 18428.41} C_VEL
LIN {X 0,Y 373.132,Z 691.617,A -85,B 0,C 180,E1 18427.968,E2 18427.968} C_VEL
LIN {X 0,Y 378.794,Z 703.609,A -85,B 0,C 180,E1 18425.02,E2 18425.02} C_VEL
LIN {X 0,Y 385.746,Z 719.455,A -85,B 0,C 180,E1 18421.489,E2 18421.489} C_VEL
LIN {X 0,Y 392.455,Z 735.856,A -85,B 0,C 180,E1 18418.174,E2 18418.174} C_VEL
LIN {X 0,Y 399.28,Z 754.006,A -85,B 0,C 180,E1 18414.835,E2 18414.835} C_VEL
LIN {X 0,Y 405.819,Z 773.44,A -85,B 0,C 180,E1 18411.584,E2 18411.584} C_VEL
LIN {X 0,Y 409.002,Z 784.098,A -85,B 0,C 180,E1 18409.925,E2 18409.925} C_VEL
LIN {X 0,Y 402.092,Z 825.75,A -85,B 0,C 180,E1 18405.675,E2 18405.675} C_VEL
LIN {X 0,Y 399.672,Z 841.352,A -85,B 0,C 180,E1 18404.087,E2 18404.087} C_VEL
LIN {X 0,Y 397.848,Z 847.754,A -85,B 0,C 180,E1 18403.513,E2 18403.513} C_VEL
LIN {X 0,Y 389.797,Z 865.269,A -85,B 0,C 180,E1 18402.205,E2 18402.205} C_VEL
LIN {X 0,Y 388.332,Z 870.774,A -85,B 0,C 180,E1 18401.694,E2 18401.694} C_VEL
LIN {X 0,Y 382.299,Z 914.802,A -85,B 0,C 180,E1 18397.17,E2 18397.17} C_VEL
LIN {X 0,Y 381.686,Z 920.657,A -85,B 0,C 180,E1 18396.61,E2 18396.61} C_VEL
LIN {X 0,Y 382.146,Z 932.928,A -85,B 0,C 180,E1 18396.159,E2 18396.159} C_VEL
LIN {X 0,Y 376.919,Z 1006.924,A -85,B 0,C 180,E1 18393.813,E2 18393.813} C_VEL
LIN {X 0,Y 373.33,Z 1064.049,A -85,B 0,C 180,E1 18391.749,E2 18391.749} C_VEL
LIN {X 0,Y 372.334,Z 1082.082,A -85,B 0,C 180,E1 18390.904,E2 18390.904} C_VEL
LIN {X 0,Y 371.069,Z 1098.921,A -85,B 0,C 180,E1 18389.817,E2 18389.817} C_VEL
LIN {X 0,Y 369.541,Z 1115.315,A -85,B 0,C 180,E1 18388.439,E2 18388.439} C_VEL
LIN {X 0,Y 367.977,Z 1130.502,A -85,B 0,C 180,E1 18386.812,E2 18386.812} C_VEL
LIN {X 0,Y 366.462,Z 1144.073,A -85,B 0,C 180,E1 18385.019,E2 18385.019} C_VEL
LIN {X 0,Y 364.98,Z 1156.986,A -85,B 0,C 180,E1 18382.894,E2 18382.894} C_VEL
LIN {X 0,Y 363.809,Z 1167.485,A -85,B 0,C 180,E1 18380.766,E2 18380.766} C_VEL
LIN {X 0,Y 362.862,Z 1177.232,A -85,B 0,C 180,E1 18378.309,E2 18378.309} C_VEL
LIN {X 0,Y 362.281,Z 1184.827,A -85,B 0,C 180,E1 18375.857,E2 18375.857} C_VEL
LIN {X 0,Y 362.035,Z 1190.973,A -85,B 0,C 180,E1 18373.252,E2 18373.252} C_VEL
LIN {X 0,Y 362.123,Z 1195.296,A -85,B 0,C 180,E1 18370.602,E2 18370.602} C_VEL
LIN {X 0,Y 362.583,Z 1197.944,A -85,B 0,C 180,E1 18367.925,E2 18367.925} C_VEL
LIN {X 0,Y 363.475,Z 1198.808,A -85,B 0,C 180,E1 18365.209,E2 18365.209} C_VEL
LIN {X 0,Y 364.88,Z 1197.971,A -85,B 0,C 180,E1 18362.513,E2 18362.513} C_VEL
LIN {X 0,Y 366.99,Z 1195.15,A -85,B 0,C 180,E1 18359.688,E2 18359.688} C_VEL
LIN {X 0,Y 369.468,Z 1190.993,A -85,B 0,C 180,E1 18357.208,E2 18357.208} C_VEL
LIN {X 0,Y 372.969,Z 1184.282,A -85,B 0,C 180,E1 18354.462,E2 18354.462} C_VEL
LIN {X 0,Y 376.71,Z 1176.325,A -85,B 0,C 180,E1 18352.067,E2 18352.067} C_VEL
LIN {X 0,Y 380.753,Z 1166.928,A -85,B 0,C 180,E1 18349.866,E2 18349.866} C_VEL
LIN {X 0,Y 385.36,Z 1155.404,A -85,B 0,C 180,E1 18347.716,E2 18347.716} C_VEL
LIN {X 0,Y 390.093,Z 1142.042,A -85,B 0,C 180,E1 18345.755,E2 18345.755} C_VEL
LIN {X 0,Y 394.791,Z 1127.5,A -85,B 0,C 180,E1 18344.05,E2 18344.05} C_VEL
LIN {X 0,Y 399.013,Z 1112.397,A -85,B 0,C 180,E1 18342.65,E2 18342.65} C_VEL
LIN {X 0,Y 402.892,Z 1096.621,A -85,B 0,C 180,E1 18341.478,E2 18341.478} C_VEL
LIN {X 0,Y 409.681,Z 1067.885,A -85,B 0,C 180,E1 18339.797,E2 18339.797} C_VEL
LIN {X 0,Y 418.527,Z 1032.702,A -85,B 0,C 180,E1 18338.118,E2 18338.118} C_VEL
LIN {X 0,Y 427.191,Z 994.868,A -85,B 0,C 180,E1 18336.598,E2 18336.598} C_VEL
LIN {X 0,Y 433.636,Z 961.316,A -85,B 0,C 180,E1 18335.432,E2 18335.432} C_VEL
LIN {X 0,Y 434.062,Z 952.757,A -85,B 0,C 180,E1 18334.703,E2 18334.703} C_VEL
LIN {X 0,Y 448.994,Z 922.749,A -85,B 0,C 180,E1 18330.956,E2 18330.956} C_VEL
LIN {X 0,Y 464.897,Z 896.661,A -85,B 0,C 180,E1 18327.619,E2 18327.619} C_VEL
LIN {X 0,Y 466.996,Z 893.574,A -85,B 0,C 180,E1 18327.218,E2 18327.218} C_VEL
LIN {X 0,Y 455.384,Z 912.452,A -85,B 0,C 180,E1 18324.762,E2 18324.762} C_VEL
LIN {X 0,Y 446.991,Z 930.016,A -85,B 0,C 180,E1 18322.252,E2 18322.252} C_VEL
LIN {X 0,Y 441.648,Z 946.396,A -85,B 0,C 180,E1 18319.723,E2 18319.723} C_VEL
LIN {X 0,Y 438.883,Z 963.123,A -85,B 0,C 180,E1 18316.994,E2 18316.994} C_VEL
LIN {X 0,Y 438.488,Z 970.548,A -85,B 0,C 180,E1 18315.77,E2 18315.77} C_VEL
LIN {X 0,Y 433.216,Z 981.254,A -85,B 0,C 180,E1 18315.286,E2 18315.286} C_VEL
LIN {X 0,Y 430.085,Z 999.534,A -85,B 0,C 180,E1 18314.921,E2 18314.921} C_VEL
LIN {X 0,Y 425.026,Z 1026.047,A -85,B 0,C 180,E1 18314.443,E2 18314.443} C_VEL
LIN {X 0,Y 420.78,Z 1046.8,A -85,B 0,C 180,E1 18313.792,E2 18313.792} C_VEL
LIN {X 0,Y 414.57,Z 1073.695,A -85,B 0,C 180,E1 18312.664,E2 18312.664} C_VEL
LIN {X 0,Y 408.342,Z 1097.335,A -85,B 0,C 180,E1 18311.383,E2 18311.383} C_VEL
LIN {X 0,Y 402.172,Z 1119.343,A -85,B 0,C 180,E1 18309.896,E2 18309.896} C_VEL
LIN {X 0,Y 395.36,Z 1142.048,A -85,B 0,C 180,E1 18308.009,E2 18308.009} C_VEL
LIN {X 0,Y 389.302,Z 1161.729,A -85,B 0,C 180,E1 18306.024,E2 18306.024} C_VEL
LIN {X 0,Y 383.366,Z 1180.551,A -85,B 0,C 180,E1 18303.745,E2 18303.745} C_VEL
LIN {X 0,Y 377.579,Z 1198.799,A -85,B 0,C 180,E1 18301.087,E2 18301.087} C_VEL
LIN {X 0,Y 372.745,Z 1214.538,A -85,B 0,C 180,E1 18298.344,E2 18298.344} C_VEL
LIN {X 0,Y 368.598,Z 1228.849,A -85,B 0,C 180,E1 18295.376,E2 18295.376} C_VEL
LIN {X 0,Y 365.157,Z 1242.209,A -85,B 0,C 180,E1 18292.03,E2 18292.03} C_VEL
LIN {X 0,Y 363.588,Z 1249.696,A -85,B 0,C 180,E1 18289.936,E2 18289.936} C_VEL
LIN {X 0,Y 361.97,Z 1261.369,A -85,B 0,C 180,E1 18286.858,E2 18286.858} C_VEL
LIN {X 0,Y 360.955,Z 1270.999,A -85,B 0,C 180,E1 18283.78,E2 18283.78} C_VEL
LIN {X 0,Y 360.453,Z 1278.33,A -85,B 0,C 180,E1 18280.87,E2 18280.87} C_VEL
LIN {X 0,Y 360.308,Z 1284.322,A -85,B 0,C 180,E1 18277.813,E2 18277.813} C_VEL
LIN {X 0,Y 360.345,Z 1288.735,A -85,B 0,C 180,E1 18274.773,E2 18274.773} C_VEL
LIN {X 0,Y 360.406,Z 1291.307,A -85,B 0,C 180,E1 18271.906,E2 18271.906} C_VEL
LIN {X 0,Y 360.367,Z 1292.655,A -85,B 0,C 180,E1 18268.885,E2 18268.885} C_VEL
LIN {X 0,Y 360.223,Z 1292.379,A -85,B 0,C 180,E1 18265.859,E2 18265.859} C_VEL
LIN {X 0,Y 360.156,Z 1290.609,A -85,B 0,C 180,E1 18262.661,E2 18262.661} C_VEL
LIN {X 0,Y 360.355,Z 1287.216,A -85,B 0,C 180,E1 18259.446,E2 18259.446} C_VEL
LIN {X 0,Y 361.158,Z 1281.979,A -85,B 0,C 180,E1 18256.06,E2 18256.06} C_VEL
LIN {X 0,Y 362.745,Z 1275.04,A -85,B 0,C 180,E1 18252.679,E2 18252.679} C_VEL
LIN {X 0,Y 365.274,Z 1266.221,A -85,B 0,C 180,E1 18249.32,E2 18249.32} C_VEL
LIN {X 0,Y 368.88,Z 1255.454,A -85,B 0,C 180,E1 18245.991,E2 18245.991} C_VEL
LIN {X 0,Y 373.847,Z 1242.169,A -85,B 0,C 180,E1 18242.609,E2 18242.609} C_VEL
LIN {X 0,Y 379.554,Z 1228.038,A -85,B 0,C 180,E1 18239.614,E2 18239.614} C_VEL
LIN {X 0,Y 386.646,Z 1211.326,A -85,B 0,C 180,E1 18236.647,E2 18236.647} C_VEL
LIN {X 0,Y 395.181,Z 1191.91,A -85,B 0,C 180,E1 18233.788,E2 18233.788} C_VEL
LIN {X 0,Y 404.462,Z 1171.391,A -85,B 0,C 180,E1 18231.283,E2 18231.283} C_VEL
LIN {X 0,Y 414.525,Z 1149.571,A -85,B 0,C 180,E1 18229.087,E2 18229.087} C_VEL
LIN {X 0,Y 424.956,Z 1127.103,A -85,B 0,C 180,E1 18227.247,E2 18227.247} C_VEL
LIN {X 0,Y 435.526,Z 1103.985,A -85,B 0,C 180,E1 18225.737,E2 18225.737} C_VEL
LIN {X 0,Y 445.664,Z 1080.794,A -85,B 0,C 180,E1 18224.573,E2 18224.573} C_VEL
LIN {X 0,Y 446.264,Z 1079.366,A -85,B 0,C 180,E1 18224.487,E2 18224.487} C_VEL
LIN {X 0,Y 436.846,Z 1100.475,A -85,B 0,C 180,E1 18223.187,E2 18223.187} C_VEL
LIN {X 0,Y 426.77,Z 1121.858,A -85,B 0,C 180,E1 18221.533,E2 18221.533} C_VEL
LIN {X 0,Y 416.778,Z 1142.504,A -85,B 0,C 180,E1 18219.566,E2 18219.566} C_VEL
LIN {X 0,Y 407.052,Z 1162.335,A -85,B 0,C 180,E1 18217.26,E2 18217.26} C_VEL
LIN {X 0,Y 398.23,Z 1180.212,A -85,B 0,C 180,E1 18214.748,E2 18214.748} C_VEL
LIN {X 0,Y 390.285,Z 1196.303,A -85,B 0,C 180,E1 18212.027,E2 18212.027} C_VEL
LIN {X 0,Y 383.407,Z 1210.296,A -85,B 0,C 180,E1 18209.188,E2 18209.188} C_VEL
LIN {X 0,Y 377.009,Z 1223.396,A -85,B 0,C 180,E1 18205.951,E2 18205.951} C_VEL
LIN {X 0,Y 371.785,Z 1234.288,A -85,B 0,C 180,E1 18202.618,E2 18202.618} C_VEL
LIN {X 0,Y 367.85,Z 1242.764,A -85,B 0,C 180,E1 18199.367,E2 18199.367} C_VEL
LIN {X 0,Y 364.761,Z 1249.816,A -85,B 0,C 180,E1 18195.91,E2 18195.91} C_VEL
LIN {X 0,Y 362.717,Z 1254.87,A -85,B 0,C 180,E1 18192.579,E2 18192.579} C_VEL
LIN {X 0,Y 361.391,Z 1258.264,A -85,B 0,C 180,E1 18189.234,E2 18189.234} C_VEL
LIN {X 0,Y 360.645,Z 1260.045,A -85,B 0,C 180,E1 18185.888,E2 18185.888} C_VEL
LIN {X 0,Y 360.303,Z 1260.324,A -85,B 0,C 180,E1 18182.704,E2 18182.704} C_VEL
LIN {X 0,Y 360.19,Z 1259.128,A -85,B 0,C 180,E1 18179.682,E2 18179.682} C_VEL
LIN {X 0,Y 360.16,Z 1256.262,A -85,B 0,C 180,E1 18176.339,E2 18176.339} C_VEL
LIN {X 0,Y 360.304,Z 1252.215,A -85,B 0,C 180,E1 18173.307,E2 18173.307} C_VEL
LIN {X 0,Y 360.701,Z 1246.212,A -85,B 0,C 180,E1 18170.103,E2 18170.103} C_VEL
LIN {X 0,Y 361.544,Z 1238.161,A -85,B 0,C 180,E1 18166.784,E2 18166.784} C_VEL
LIN {X 0,Y 362.826,Z 1228.75,A -85,B 0,C 180,E1 18163.674,E2 18163.674} C_VEL
LIN {X 0,Y 364.685,Z 1217.409,A -85,B 0,C 180,E1 18160.595,E2 18160.595} C_VEL
LIN {X 0,Y 366.981,Z 1204.72,A -85,B 0,C 180,E1 18157.745,E2 18157.745} C_VEL
LIN {X 0,Y 369.728,Z 1190.507,A -85,B 0,C 180,E1 18155.046,E2 18155.046} C_VEL
LIN {X 0,Y 372.946,Z 1174.373,A -85,B 0,C 180,E1 18152.452,E2 18152.452} C_VEL
LIN {X 0,Y 376.357,Z 1157.273,A -85,B 0,C 180,E1 18150.123,E2 18150.123} C_VEL
LIN {X 0,Y 379.958,Z 1138.631,A -85,B 0,C 180,E1 18147.977,E2 18147.977} C_VEL
LIN {X 0,Y 383.676,Z 1118.192,A -85,B 0,C 180,E1 18146.013,E2 18146.013} C_VEL
LIN {X 0,Y 387.109,Z 1097.713,A -85,B 0,C 180,E1 18144.376,E2 18144.376} C_VEL
LIN {X 0,Y 390.281,Z 1076.629,A -85,B 0,C 180,E1 18142.982,E2 18142.982} C_VEL
LIN {X 0,Y 393.215,Z 1054.375,A -85,B 0,C 180,E1 18141.791,E2 18141.791} C_VEL
LIN {X 0,Y 395.749,Z 1031.35,A -85,B 0,C 180,E1 18140.828,E2 18140.828} C_VEL
LIN {X 0,Y 397.825,Z 1006.904,A -85,B 0,C 180,E1 18140.081,E2 18140.081} C_VEL
LIN {X 0,Y 413.86,Z 787.152,A -85,B 0,C 180,E1 18134.892,E2 18134.892} C_VEL
LIN {X 0,Y 398.495,Z 756.924,A -85,B 0,C 180,E1 18132.332,E2 18132.332} C_VEL
LIN {X 0,Y 383.262,Z 729.086,A -85,B 0,C 180,E1 18129.611,E2 18129.611} C_VEL
LIN {X 0,Y 373.175,Z 711.574,A -85,B 0,C 180,E1 18127.657,E2 18127.657} C_VEL
LIN {X 0,Y 366.043,Z 694.857,A -85,B 0,C 180,E1 18124.435,E2 18124.435} C_VEL
LIN {X 0,Y 363.019,Z 687.756,A -85,B 0,C 180,E1 18123.018,E2 18123.018} C_VEL
LIN {X 0,Y 362.976,Z 687.453,A -85,B 0,C 180,E1 18122.84,E2 18122.84} C_VEL
LIN {X 0,Y 362.97,Z 687.455,A -85,B 0,C 180,E1 18118.643,E2 18118.643} C_VEL
LIN {X 0,Y 362.965,Z 687.455,A -85,B 0,C 180,E1 18114.409,E2 18114.409} C_VEL
LIN {X 0,Y 362.978,Z 687.455,A -85,B 0,C 180,E1 18110.143,E2 18110.143} C_VEL
LIN {X 0,Y 362.965,Z 687.456,A -85,B 0,C 180,E1 18105.966,E2 18105.966} C_VEL
LIN {X 0,Y 362.963,Z 687.448,A -85,B 0,C 180,E1 18101.764,E2 18101.764} C_VEL
LIN {X 0,Y 362.978,Z 687.439,A -85,B 0,C 180,E1 18097.6,E2 18097.6} C_VEL
LIN {X 0,Y 362.962,Z 687.442,A -85,B 0,C 180,E1 18093.477,E2 18093.477} C_VEL
LIN {X 0,Y 362.962,Z 687.442,A -85,B 0,C 180,E1 18089.371,E2 18089.371} C_VEL
LIN {X 0,Y 362.971,Z 687.444,A -85,B 0,C 180,E1 18085.103,E2 18085.103} C_VEL
LIN {X 0,Y 362.964,Z 687.453,A -85,B 0,C 180,E1 18080.968,E2 18080.968} C_VEL
LIN {X 0,Y 362.965,Z 687.455,A -85,B 0,C 180,E1 18076.785,E2 18076.785} C_VEL
LIN {X 0,Y 362.974,Z 687.447,A -85,B 0,C 180,E1 18072.694,E2 18072.694} C_VEL
LIN {X 0,Y 362.995,Z 687.621,A -85,B 0,C 180,E1 18070.659,E2 18070.659} C_VEL
LIN {X 0,Y 364.357,Z 691.059,A -85,B 0,C 180,E1 18069.773,E2 18069.773} C_VEL
LIN {X 0,Y 365.229,Z 692.645,A -85,B 0,C 180,E1 18069.322,E2 18069.322} C_VEL
LIN {X 0,Y 371.082,Z 704.971,A -85,B 0,C 180,E1 18066.163,E2 18066.163} C_VEL
LIN {X 0,Y 377.652,Z 719.657,A -85,B 0,C 180,E1 18062.742,E2 18062.742} C_VEL
LIN {X 0,Y 384.611,Z 736.538,A -85,B 0,C 180,E1 18059.196,E2 18059.196} C_VEL
LIN {X 0,Y 391.357,Z 754.373,A -85,B 0,C 180,E1 18055.803,E2 18055.803} C_VEL
LIN {X 0,Y 397.802,Z 773.226,A -85,B 0,C 180,E1 18052.538,E2 18052.538} C_VEL
LIN {X 0,Y 401.98,Z 786.91,A -85,B 0,C 180,E1 18050.35,E2 18050.35} C_VEL
LIN {X 0,Y 394.894,Z 828.305,A -85,B 0,C 180,E1 18046.074,E2 18046.074} C_VEL
LIN {X 0,Y 388.332,Z 870.774,A -85,B 0,C 180,E1 18041.694,E2 18041.694} C_VEL
LIN {X 0,Y 386.534,Z 877.206,A -85,B 0,C 180,E1 18041.105,E2 18041.105} C_VEL
LIN {X 0,Y 378.499,Z 894.716,A -85,B 0,C 180,E1 18039.756,E2 18039.756} C_VEL
LIN {X 0,Y 377.045,Z 900.236,A -85,B 0,C 180,E1 18039.235,E2 18039.235} C_VEL
LIN {X 0,Y 374.326,Z 921.2,A -85,B 0,C 180,E1 18037.087,E2 18037.087} C_VEL
LIN {X 0,Y 374.765,Z 933.516,A -85,B 0,C 180,E1 18036.624,E2 18036.624} C_VEL
LIN {X 0,Y 369.094,Z 1010.936,A -85,B 0,C 180,E1 18034.086,E2 18034.086} C_VEL
LIN {X 0,Y 365.567,Z 1065.896,A -85,B 0,C 180,E1 18032.028,E2 18032.028} C_VEL
LIN {X 0,Y 364.531,Z 1083.662,A -85,B 0,C 180,E1 18031.158,E2 18031.158} C_VEL
LIN {X 0,Y 363.253,Z 1100.055,A -85,B 0,C 180,E1 18030.065,E2 18030.065} C_VEL
LIN {X 0,Y 361.692,Z 1116.259,A -85,B 0,C 180,E1 18028.662,E2 18028.662} C_VEL
LIN {X 0,Y 360.164,Z 1130.655,A -85,B 0,C 180,E1 18027.084,E2 18027.084} C_VEL
LIN {X 0,Y 358.538,Z 1144.859,A -85,B 0,C 180,E1 18025.169,E2 18025.169} C_VEL
LIN {X 0,Y 356.969,Z 1158.25,A -85,B 0,C 180,E1 18022.914,E2 18022.914} C_VEL
LIN {X 0,Y 355.74,Z 1169.181,A -85,B 0,C 180,E1 18020.623,E2 18020.623} C_VEL
LIN {X 0,Y 354.851,Z 1178.409,A -85,B 0,C 180,E1 18018.227,E2 18018.227} C_VEL
LIN {X 0,Y 354.256,Z 1186.412,A -85,B 0,C 180,E1 18015.554,E2 18015.554} C_VEL
LIN {X 0,Y 354.057,Z 1192.384,A -85,B 0,C 180,E1 18012.891,E2 18012.891} C_VEL
LIN {X 0,Y 354.246,Z 1196.933,A -85,B 0,C 180,E1 18009.915,E2 18009.915} C_VEL
LIN {X 0,Y 354.843,Z 1199.3,A -85,B 0,C 180,E1 18007.122,E2 18007.122} C_VEL
LIN {X 0,Y 355.947,Z 1199.923,A -85,B 0,C 180,E1 18004.309,E2 18004.309} C_VEL
LIN {X 0,Y 357.664,Z 1198.647,A -85,B 0,C 180,E1 18001.442,E2 18001.442} C_VEL
LIN {X 0,Y 359.961,Z 1195.697,A -85,B 0,C 180,E1 17998.727,E2 17998.727} C_VEL
LIN {X 0,Y 363.12,Z 1190.618,A -85,B 0,C 180,E1 17995.894,E2 17995.894} C_VEL
LIN {X 0,Y 366.819,Z 1183.819,A -85,B 0,C 180,E1 17993.269,E2 17993.269} C_VEL
LIN {X 0,Y 370.935,Z 1175.491,A -85,B 0,C 180,E1 17990.849,E2 17990.849} C_VEL
LIN {X 0,Y 375.377,Z 1165.76,A -85,B 0,C 180,E1 17988.632,E2 17988.632} C_VEL
LIN {X 0,Y 380.336,Z 1153.668,A -85,B 0,C 180,E1 17986.469,E2 17986.469} C_VEL
LIN {X 0,Y 384.91,Z 1141.492,A -85,B 0,C 180,E1 17984.712,E2 17984.712} C_VEL
LIN {X 0,Y 389.692,Z 1127.306,A -85,B 0,C 180,E1 17983.069,E2 17983.069} C_VEL
LIN {X 0,Y 394.212,Z 1112.295,A -85,B 0,C 180,E1 17981.668,E2 17981.668} C_VEL
LIN {X 0,Y 398.801,Z 1094.509,A -85,B 0,C 180,E1 17980.368,E2 17980.368} C_VEL
LIN {X 0,Y 406.735,Z 1063.802,A -85,B 0,C 180,E1 17978.588,E2 17978.588} C_VEL
LIN {X 0,Y 416.375,Z 1027.352,A -85,B 0,C 180,E1 17976.881,E2 17976.881} C_VEL
LIN {X 0,Y 425.018,Z 990.29,A -85,B 0,C 180,E1 17975.429,E2 17975.429} C_VEL
LIN {X 0,Y 430.265,Z 963.825,A -85,B 0,C 180,E1 17974.51,E2 17974.51} C_VEL
LIN {X 0,Y 430.829,Z 954.364,A -85,B 0,C 180,E1 17973.686,E2 17973.686} C_VEL
LIN {X 0,Y 446.733,Z 924.516,A -85,B 0,C 180,E1 17969.91,E2 17969.91} C_VEL
LIN {X 0,Y 459.977,Z 903.789,A -85,B 0,C 180,E1 17967.216,E2 17967.216} C_VEL
LIN {X 0,Y 448.998,Z 921.834,A -85,B 0,C 180,E1 17964.776,E2 17964.776} C_VEL
LIN {X 0,Y 441.033,Z 938.782,A -85,B 0,C 180,E1 17962.256,E2 17962.256} C_VEL
LIN {X 0,Y 435.818,Z 955.285,A -85,B 0,C 180,E1 17959.611,E2 17959.611} C_VEL
LIN {X 0,Y 433.423,Z 971.142,A -85,B 0,C 180,E1 17956.932,E2 17956.932} C_VEL
LIN {X 0,Y 433.285,Z 973.217,A -85,B 0,C 180,E1 17956.577,E2 17956.577} C_VEL
LIN {X 0,Y 430.037,Z 979.849,A -85,B 0,C 180,E1 17956.284,E2 17956.284} C_VEL
LIN {X 0,Y 426.696,Z 999.086,A -85,B 0,C 180,E1 17955.891,E2 17955.891} C_VEL
LIN {X 0,Y 421.499,Z 1025.058,A -85,B 0,C 180,E1 17955.428,E2 17955.428} C_VEL
LIN {X 0,Y 417.113,Z 1045.154,A -85,B 0,C 180,E1 17954.807,E2 17954.807} C_VEL
LIN {X 0,Y 410.834,Z 1071.257,A -85,B 0,C 180,E1 17953.722,E2 17953.722} C_VEL
LIN {X 0,Y 403.741,Z 1096.834,A -85,B 0,C 180,E1 17952.344,E2 17952.344} C_VEL
LIN {X 0,Y 397.291,Z 1118.486,A -85,B 0,C 180,E1 17950.868,E2 17950.868} C_VEL
LIN {X 0,Y 389.942,Z 1141.78,A -85,B 0,C 180,E1 17948.916,E2 17948.916} C_VEL
LIN {X 0,Y 383.154,Z 1162.427,A -85,B 0,C 180,E1 17946.789,E2 17946.789} C_VEL
LIN {X 0,Y 377.114,Z 1180.313,A -85,B 0,C 180,E1 17944.566,E2 17944.566} C_VEL
LIN {X 0,Y 371.324,Z 1197.424,A -85,B 0,C 180,E1 17942.035,E2 17942.035} C_VEL
LIN {X 0,Y 366.121,Z 1213.125,A -85,B 0,C 180,E1 17939.262,E2 17939.262} C_VEL
LIN {X 0,Y 361.413,Z 1228.077,A -85,B 0,C 180,E1 17936.094,E2 17936.094} C_VEL
LIN {X 0,Y 357.852,Z 1240.751,A -85,B 0,C 180,E1 17932.851,E2 17932.851} C_VEL
LIN {X 0,Y 355.136,Z 1252.733,A -85,B 0,C 180,E1 17929.231,E2 17929.231} C_VEL
LIN {X 0,Y 353.706,Z 1263.326,A -85,B 0,C 180,E1 17926.249,E2 17926.249} C_VEL
LIN {X 0,Y 352.85,Z 1272.029,A -85,B 0,C 180,E1 17923.267,E2 17923.267} C_VEL
LIN {X 0,Y 352.41,Z 1279.528,A -85,B 0,C 180,E1 17920.087,E2 17920.087} C_VEL
LIN {X 0,Y 352.34,Z 1285.06,A -85,B 0,C 180,E1 17917.007,E2 17917.007} C_VEL
LIN {X 0,Y 352.393,Z 1289.006,A -85,B 0,C 180,E1 17913.902,E2 17913.902} C_VEL
LIN {X 0,Y 352.434,Z 1291.329,A -85,B 0,C 180,E1 17910.973,E2 17910.973} C_VEL
LIN {X 0,Y 352.336,Z 1292.219,A -85,B 0,C 180,E1 17907.884,E2 17907.884} C_VEL
LIN {X 0,Y 352.186,Z 1291.744,A -85,B 0,C 180,E1 17904.949,E2 17904.949} C_VEL
LIN {X 0,Y 352.168,Z 1289.646,A -85,B 0,C 180,E1 17901.672,E2 17901.672} C_VEL
LIN {X 0,Y 352.56,Z 1285.851,A -85,B 0,C 180,E1 17898.215,E2 17898.215} C_VEL
LIN {X 0,Y 353.662,Z 1280.249,A -85,B 0,C 180,E1 17894.754,E2 17894.754} C_VEL
LIN {X 0,Y 355.775,Z 1272.558,A -85,B 0,C 180,E1 17891.141,E2 17891.141} C_VEL
LIN {X 0,Y 359.015,Z 1262.917,A -85,B 0,C 180,E1 17887.568,E2 17887.568} C_VEL
LIN {X 0,Y 363.441,Z 1251.438,A -85,B 0,C 180,E1 17884.111,E2 17884.111} C_VEL
LIN {X 0,Y 369.056,Z 1238.056,A -85,B 0,C 180,E1 17880.81,E2 17880.81} C_VEL
LIN {X 0,Y 375.877,Z 1222.786,A -85,B 0,C 180,E1 17877.675,E2 17877.675} C_VEL
LIN {X 0,Y 384.065,Z 1205.312,A -85,B 0,C 180,E1 17874.691,E2 17874.691} C_VEL
LIN {X 0,Y 393.663,Z 1185.554,A -85,B 0,C 180,E1 17871.886,E2 17871.886} C_VEL
LIN {X 0,Y 404.249,Z 1164.394,A -85,B 0,C 180,E1 17869.418,E2 17869.418} C_VEL
LIN {X 0,Y 415.366,Z 1142.562,A -85,B 0,C 180,E1 17867.339,E2 17867.339} C_VEL
LIN {X 0,Y 426.788,Z 1120.146,A -85,B 0,C 180,E1 17865.625,E2 17865.625} C_VEL
LIN {X 0,Y 436.947,Z 1099.764,A -85,B 0,C 180,E1 17864.384,E2 17864.384} C_VEL
LIN {X 0,Y 426.076,Z 1120.943,A -85,B 0,C 180,E1 17862.796,E2 17862.796} C_VEL
LIN {X 0,Y 414.894,Z 1142.008,A -85,B 0,C 180,E1 17860.821,E2 17860.821} C_VEL
LIN {X 0,Y 404.334,Z 1161.651,A -85,B 0,C 180,E1 17858.549,E2 17858.549} C_VEL
LIN {X 0,Y 394.563,Z 1179.75,A -85,B 0,C 180,E1 17856.01,E2 17856.01} C_VEL
LIN {X 0,Y 385.573,Z 1196.393,A -85,B 0,C 180,E1 17853.174,E2 17853.174} C_VEL
LIN {X 0,Y 377.796,Z 1210.885,A -85,B 0,C 180,E1 17850.19,E2 17850.19} C_VEL
LIN {X 0,Y 370.904,Z 1223.819,A -85,B 0,C 180,E1 17846.93,E2 17846.93} C_VEL
LIN {X 0,Y 365.228,Z 1234.616,A -85,B 0,C 180,E1 17843.56,E2 17843.56} C_VEL
LIN {X 0,Y 360.912,Z 1243.068,A -85,B 0,C 180,E1 17840.262,E2 17840.262} C_VEL
LIN {X 0,Y 357.358,Z 1250.401,A -85,B 0,C 180,E1 17836.583,E2 17836.583} C_VEL
LIN {X 0,Y 354.994,Z 1255.584,A -85,B 0,C 180,E1 17833.022,E2 17833.022} C_VEL
LIN {X 0,Y 353.494,Z 1259.034,A -85,B 0,C 180,E1 17829.443,E2 17829.443} C_VEL
LIN {X 0,Y 352.687,Z 1260.617,A -85,B 0,C 180,E1 17826.021,E2 17826.021} C_VEL
LIN {X 0,Y 352.303,Z 1260.664,A -85,B 0,C 180,E1 17822.603,E2 17822.603} C_VEL
LIN {X 0,Y 352.188,Z 1259.235,A -85,B 0,C 180,E1 17819.349,E2 17819.349} C_VEL
LIN {X 0,Y 352.166,Z 1256.183,A -85,B 0,C 180,E1 17816.093,E2 17816.093} C_VEL
LIN {X 0,Y 352.352,Z 1251.603,A -85,B 0,C 180,E1 17812.827,E2 17812.827} C_VEL
LIN {X 0,Y 352.814,Z 1245.349,A -85,B 0,C 180,E1 17809.55,E2 17809.55} C_VEL
LIN {X 0,Y 353.656,Z 1237.613,A -85,B 0,C 180,E1 17806.428,E2 17806.428} C_VEL
LIN {X 0,Y 355.083,Z 1227.561,A -85,B 0,C 180,E1 17803.139,E2 17803.139} C_VEL
LIN {X 0,Y 356.929,Z 1216.649,A -85,B 0,C 180,E1 17800.186,E2 17800.186} C_VEL
LIN {X 0,Y 359.367,Z 1203.666,A -85,B 0,C 180,E1 17797.247,E2 17797.247} C_VEL
LIN {X 0,Y 362.247,Z 1189.147,A -85,B 0,C 180,E1 17794.494,E2 17794.494} C_VEL
LIN {X 0,Y 365.491,Z 1173.203,A -85,B 0,C 180,E1 17791.93,E2 17791.93} C_VEL
LIN {X 0,Y 369.192,Z 1155.004,A -85,B 0,C 180,E1 17789.459,E2 17789.459} C_VEL
LIN {X 0,Y 372.904,Z 1136.066,A -85,B 0,C 180,E1 17787.296,E2 17787.296} C_VEL
LIN {X 0,Y 376.617,Z 1116.074,A -85,B 0,C 180,E1 17785.378,E2 17785.378} C_VEL
LIN {X 0,Y 380.171,Z 1095.208,A -85,B 0,C 180,E1 17783.717,E2 17783.717} C_VEL
LIN {X 0,Y 383.454,Z 1073.513,A -85,B 0,C 180,E1 17782.303,E2 17782.303} C_VEL
LIN {X 0,Y 386.39,Z 1051.159,A -85,B 0,C 180,E1 17781.131,E2 17781.131} C_VEL
LIN {X 0,Y 389.005,Z 1026.836,A -85,B 0,C 180,E1 17780.146,E2 17780.146} C_VEL
LIN {X 0,Y 391.212,Z 1000.2,A -85,B 0,C 180,E1 17779.376,E2 17779.376} C_VEL
LIN {X 0,Y 407.095,Z 789.725,A -85,B 0,C 180,E1 17774.298,E2 17774.298} C_VEL
LIN {X 0,Y 392.068,Z 760.135,A -85,B 0,C 180,E1 17771.732,E2 17771.732} C_VEL
LIN {X 0,Y 377.07,Z 732.656,A -85,B 0,C 180,E1 17768.987,E2 17768.987} C_VEL
LIN {X 0,Y 365.195,Z 712.2,A -85,B 0,C 180,E1 17766.648,E2 17766.648} C_VEL
LIN {X 0,Y 358.461,Z 696.4,A -85,B 0,C 180,E1 17763.527,E2 17763.527} C_VEL
LIN {X 0,Y 355.1,Z 688.909,A -85,B 0,C 180,E1 17761.965,E2 17761.965} C_VEL
LIN {X 0,Y 355.025,Z 688.438,A -85,B 0,C 180,E1 17761.852,E2 17761.852} C_VEL
LIN {X 0,Y 355.028,Z 688.442,A -85,B 0,C 180,E1 17757.693,E2 17757.693} C_VEL
LIN {X 0,Y 355.039,Z 688.443,A -85,B 0,C 180,E1 17753.399,E2 17753.399} C_VEL
LIN {X 0,Y 355.028,Z 688.44,A -85,B 0,C 180,E1 17749.071,E2 17749.071} C_VEL
LIN {X 0,Y 355.031,Z 688.441,A -85,B 0,C 180,E1 17744.852,E2 17744.852} C_VEL
LIN {X 0,Y 355.033,Z 688.444,A -85,B 0,C 180,E1 17740.609,E2 17740.609} C_VEL
LIN {X 0,Y 355.034,Z 688.444,A -85,B 0,C 180,E1 17736.308,E2 17736.308} C_VEL
LIN {X 0,Y 355.027,Z 688.445,A -85,B 0,C 180,E1 17732.1,E2 17732.1} C_VEL
LIN {X 0,Y 355.032,Z 688.445,A -85,B 0,C 180,E1 17728.065,E2 17728.065} C_VEL
LIN {X 0,Y 355.034,Z 688.445,A -85,B 0,C 180,E1 17723.808,E2 17723.808} C_VEL
LIN {X 0,Y 355.025,Z 688.436,A -85,B 0,C 180,E1 17719.618,E2 17719.618} C_VEL
LIN {X 0,Y 355.042,Z 688.433,A -85,B 0,C 180,E1 17715.487,E2 17715.487} C_VEL
LIN {X 0,Y 355.037,Z 688.48,A -85,B 0,C 180,E1 17712.202,E2 17712.202} C_VEL
LIN {X 0,Y 356.22,Z 691.751,A -85,B 0,C 180,E1 17711.34,E2 17711.34} C_VEL
LIN {X 0,Y 357.37,Z 693.814,A -85,B 0,C 180,E1 17710.725,E2 17710.725} C_VEL
LIN {X 0,Y 361.464,Z 702.292,A -85,B 0,C 180,E1 17708.416,E2 17708.416} C_VEL
LIN {X 0,Y 367.054,Z 714.387,A -85,B 0,C 180,E1 17705.371,E2 17705.371} C_VEL
LIN {X 0,Y 373.336,Z 728.839,A -85,B 0,C 180,E1 17702.053,E2 17702.053} C_VEL
LIN {X 0,Y 379.967,Z 745.453,A -85,B 0,C 180,E1 17698.601,E2 17698.601} C_VEL
LIN {X 0,Y 386.679,Z 763.775,A -85,B 0,C 180,E1 17695.15,E2 17695.15} C_VEL
LIN {X 0,Y 392.745,Z 782.338,A -85,B 0,C 180,E1 17691.971,E2 17691.971} C_VEL
LIN {X 0,Y 394.944,Z 789.76,A -85,B 0,C 180,E1 17690.779,E2 17690.779} C_VEL
LIN {X 0,Y 387.655,Z 831.159,A -85,B 0,C 180,E1 17686.452,E2 17686.452} C_VEL
LIN {X 0,Y 380.91,Z 873.572,A -85,B 0,C 180,E1 17682.019,E2 17682.019} C_VEL
LIN {X 0,Y 377.045,Z 900.236,A -85,B 0,C 180,E1 17679.235,E2 17679.235} C_VEL
LIN {X 0,Y 375.531,Z 904.588,A -85,B 0,C 180,E1 17678.855,E2 17678.855} C_VEL
LIN {X 0,Y 368.343,Z 916.118,A -85,B 0,C 180,E1 17678.089,E2 17678.089} C_VEL
LIN {X 0,Y 367.15,Z 919.853,A -85,B 0,C 180,E1 17677.748,E2 17677.748} C_VEL
LIN {X 0,Y 366.994,Z 922.266,A -85,B 0,C 180,E1 17677.553,E2 17677.553} C_VEL
LIN {X 0,Y 367.363,Z 934.23,A -85,B 0,C 180,E1 17677.09,E2 17677.09} C_VEL
LIN {X 0,Y 361.59,Z 1010.613,A -85,B 0,C 180,E1 17674.522,E2 17674.522} C_VEL
LIN {X 0,Y 357.917,Z 1065.633,A -85,B 0,C 180,E1 17672.404,E2 17672.404} C_VEL
LIN {X 0,Y 356.827,Z 1083.697,A -85,B 0,C 180,E1 17671.501,E2 17671.501} C_VEL
LIN {X 0,Y 355.541,Z 1099.807,A -85,B 0,C 180,E1 17670.412,E2 17670.412} C_VEL
LIN {X 0,Y 353.842,Z 1116.989,A -85,B 0,C 180,E1 17668.896,E2 17668.896} C_VEL
LIN {X 0,Y 352.201,Z 1132.095,A -85,B 0,C 180,E1 17667.199,E2 17667.199} C_VEL
LIN {X 0,Y 350.602,Z 1145.747,A -85,B 0,C 180,E1 17665.31,E2 17665.31} C_VEL
LIN {X 0,Y 349.066,Z 1158.601,A -85,B 0,C 180,E1 17663.106,E2 17663.106} C_VEL
LIN {X 0,Y 347.856,Z 1169.182,A -85,B 0,C 180,E1 17660.881,E2 17660.881} C_VEL
LIN {X 0,Y 346.886,Z 1178.953,A -85,B 0,C 180,E1 17658.312,E2 17658.312} C_VEL
LIN {X 0,Y 346.304,Z 1186.613,A -85,B 0,C 180,E1 17655.748,E2 17655.748} C_VEL
LIN {X 0,Y 346.084,Z 1193.155,A -85,B 0,C 180,E1 17652.854,E2 17652.854} C_VEL
LIN {X 0,Y 346.273,Z 1197.6,A -85,B 0,C 180,E1 17649.977,E2 17649.977} C_VEL
LIN {X 0,Y 346.892,Z 1200.23,A -85,B 0,C 180,E1 17647.12,E2 17647.12} C_VEL
LIN {X 0,Y 348.096,Z 1201.049,A -85,B 0,C 180,E1 17644.118,E2 17644.118} C_VEL
LIN {X 0,Y 349.824,Z 1200.045,A -85,B 0,C 180,E1 17641.31,E2 17641.31} C_VEL
LIN {X 0,Y 352.382,Z 1197.158,A -85,B 0,C 180,E1 17638.374,E2 17638.374} C_VEL
LIN {X 0,Y 355.706,Z 1192.245,A -85,B 0,C 180,E1 17635.486,E2 17635.486} C_VEL
LIN {X 0,Y 359.344,Z 1186.111,A -85,B 0,C 180,E1 17632.967,E2 17632.967} C_VEL
LIN {X 0,Y 363.922,Z 1177.65,A -85,B 0,C 180,E1 17630.352,E2 17630.352} C_VEL
LIN {X 0,Y 369.209,Z 1166.731,A -85,B 0,C 180,E1 17627.805,E2 17627.805} C_VEL
LIN {X 0,Y 374.484,Z 1154.784,A -85,B 0,C 180,E1 17625.622,E2 17625.622} C_VEL
LIN {X 0,Y 379.916,Z 1141.049,A -85,B 0,C 180,E1 17623.644,E2 17623.644} C_VEL
LIN {X 0,Y 385.015,Z 1126.707,A -85,B 0,C 180,E1 17621.998,E2 17621.998} C_VEL
LIN {X 0,Y 390.051,Z 1110.733,A -85,B 0,C 180,E1 17620.534,E2 17620.534} C_VEL
LIN {X 0,Y 395.248,Z 1091.753,A -85,B 0,C 180,E1 17619.18,E2 17619.18} C_VEL
LIN {X 0,Y 403.953,Z 1060.802,A -85,B 0,C 180,E1 17617.402,E2 17617.402} C_VEL
LIN {X 0,Y 414.173,Z 1023.711,A -85,B 0,C 180,E1 17615.693,E2 17615.693} C_VEL
LIN {X 0,Y 422.755,Z 987.754,A -85,B 0,C 180,E1 17614.311,E2 17614.311} C_VEL
LIN {X 0,Y 427.1,Z 966.362,A -85,B 0,C 180,E1 17613.57,E2 17613.57} C_VEL
LIN {X 0,Y 428.11,Z 955.782,A -85,B 0,C 180,E1 17612.606,E2 17612.606} C_VEL
LIN {X 0,Y 443.153,Z 929.046,A -85,B 0,C 180,E1 17609.191,E2 17609.191} C_VEL
LIN {X 0,Y 453.101,Z 913.84,A -85,B 0,C 180,E1 17607.218,E2 17607.218} C_VEL
LIN {X 0,Y 442.582,Z 931.339,A -85,B 0,C 180,E1 17604.752,E2 17604.752} C_VEL
LIN {X 0,Y 434.825,Z 948.298,A -85,B 0,C 180,E1 17602.122,E2 17602.122} C_VEL
LIN {X 0,Y 430.072,Z 964.175,A -85,B 0,C 180,E1 17599.483,E2 17599.483} C_VEL
LIN {X 0,Y 428.195,Z 976.254,A -85,B 0,C 180,E1 17597.401,E2 17597.401} C_VEL
LIN {X 0,Y 427.204,Z 978.984,A -85,B 0,C 180,E1 17597.304,E2 17597.304} C_VEL
LIN {X 0,Y 423.569,Z 998.792,A -85,B 0,C 180,E1 17596.885,E2 17596.885} C_VEL
LIN {X 0,Y 418.227,Z 1024.222,A -85,B 0,C 180,E1 17596.434,E2 17596.434} C_VEL
LIN {X 0,Y 413.304,Z 1045.557,A -85,B 0,C 180,E1 17595.779,E2 17595.779} C_VEL
LIN {X 0,Y 406.968,Z 1070.368,A -85,B 0,C 180,E1 17594.738,E2 17594.738} C_VEL
LIN {X 0,Y 399.304,Z 1096.703,A -85,B 0,C 180,E1 17593.32,E2 17593.32} C_VEL
LIN {X 0,Y 392.037,Z 1119.566,A -85,B 0,C 180,E1 17591.731,E2 17591.731} C_VEL
LIN {X 0,Y 384.901,Z 1141,A -85,B 0,C 180,E1 17589.912,E2 17589.912} C_VEL
LIN {X 0,Y 377.325,Z 1162.725,A -85,B 0,C 180,E1 17587.645,E2 17587.645} C_VEL
LIN {X 0,Y 369.995,Z 1182.995,A -85,B 0,C 180,E1 17585.031,E2 17585.031} C_VEL
LIN {X 0,Y 363.874,Z 1199.867,A -85,B 0,C 180,E1 17582.398,E2 17582.398} C_VEL
LIN {X 0,Y 358.243,Z 1215.766,A -85,B 0,C 180,E1 17579.419,E2 17579.419} C_VEL
LIN {X 0,Y 353.445,Z 1230.1,A -85,B 0,C 180,E1 17576.185,E2 17576.185} C_VEL
LIN {X 0,Y 349.513,Z 1243.328,A -85,B 0,C 180,E1 17572.538,E2 17572.538} C_VEL
LIN {X 0,Y 346.795,Z 1254.951,A -85,B 0,C 180,E1 17568.663,E2 17568.663} C_VEL
LIN {X 0,Y 345.373,Z 1266.078,A -85,B 0,C 180,E1 17565.273,E2 17565.273} C_VEL
LIN {X 0,Y 344.639,Z 1274.67,A -85,B 0,C 180,E1 17562.055,E2 17562.055} C_VEL
LIN {X 0,Y 344.371,Z 1281.039,A -85,B 0,C 180,E1 17559.018,E2 17559.018} C_VEL
LIN {X 0,Y 344.372,Z 1286.103,A -85,B 0,C 180,E1 17555.83,E2 17555.83} C_VEL
LIN {X 0,Y 344.442,Z 1289.403,A -85,B 0,C 180,E1 17552.826,E2 17552.826} C_VEL
LIN {X 0,Y 344.428,Z 1291.314,A -85,B 0,C 180,E1 17549.665,E2 17549.665} C_VEL
LIN {X 0,Y 344.283,Z 1291.76,A -85,B 0,C 180,E1 17546.668,E2 17546.668} C_VEL
LIN {X 0,Y 344.14,Z 1290.67,A -85,B 0,C 180,E1 17543.324,E2 17543.324} C_VEL
LIN {X 0,Y 344.295,Z 1288.033,A -85,B 0,C 180,E1 17539.905,E2 17539.905} C_VEL
LIN {X 0,Y 345.035,Z 1283.612,A -85,B 0,C 180,E1 17536.422,E2 17536.422} C_VEL
LIN {X 0,Y 346.755,Z 1277.042,A -85,B 0,C 180,E1 17532.643,E2 17532.643} C_VEL
LIN {X 0,Y 349.512,Z 1268.911,A -85,B 0,C 180,E1 17529.045,E2 17529.045} C_VEL
LIN {X 0,Y 353.553,Z 1258.617,A -85,B 0,C 180,E1 17525.433,E2 17525.433} C_VEL
LIN {X 0,Y 358.66,Z 1246.91,A -85,B 0,C 180,E1 17522.07,E2 17522.07} C_VEL
LIN {X 0,Y 365.41,Z 1232.631,A -85,B 0,C 180,E1 17518.672,E2 17518.672} C_VEL
LIN {X 0,Y 373.642,Z 1216.164,A -85,B 0,C 180,E1 17515.434,E2 17515.434} C_VEL
LIN {X 0,Y 382.952,Z 1198.33,A -85,B 0,C 180,E1 17512.527,E2 17512.527} C_VEL
LIN {X 0,Y 393.434,Z 1178.922,A -85,B 0,C 180,E1 17509.905,E2 17509.905} C_VEL
LIN {X 0,Y 404.894,Z 1158.24,A -85,B 0,C 180,E1 17507.608,E2 17507.608} C_VEL
LIN {X 0,Y 417.069,Z 1136.487,A -85,B 0,C 180,E1 17505.664,E2 17505.664} C_VEL
LIN {X 0,Y 427.547,Z 1117.535,A -85,B 0,C 180,E1 17504.275,E2 17504.275} C_VEL
LIN {X 0,Y 415.601,Z 1138.197,A -85,B 0,C 180,E1 17502.443,E2 17502.443} C_VEL
LIN {X 0,Y 403.921,Z 1158.047,A -85,B 0,C 180,E1 17500.248,E2 17500.248} C_VEL
LIN {X 0,Y 393.211,Z 1176.162,A -85,B 0,C 180,E1 17497.795,E2 17497.795} C_VEL
LIN {X 0,Y 383.267,Z 1193.005,A -85,B 0,C 180,E1 17495.026,E2 17495.026} C_VEL
LIN {X 0,Y 374.606,Z 1207.739,A -85,B 0,C 180,E1 17492.084,E2 17492.084} C_VEL
LIN {X 0,Y 366.831,Z 1221.057,A -85,B 0,C 180,E1 17488.846,E2 17488.846} C_VEL
LIN {X 0,Y 360.352,Z 1232.317,A -85,B 0,C 180,E1 17485.473,E2 17485.473} C_VEL
LIN {X 0,Y 355.121,Z 1241.649,A -85,B 0,C 180,E1 17481.992,E2 17481.992} C_VEL
LIN {X 0,Y 350.917,Z 1249.41,A -85,B 0,C 180,E1 17478.266,E2 17478.266} C_VEL
LIN {X 0,Y 347.901,Z 1255.162,A -85,B 0,C 180,E1 17474.48,E2 17474.48} C_VEL
LIN {X 0,Y 346.009,Z 1258.88,A -85,B 0,C 180,E1 17470.827,E2 17470.827} C_VEL
LIN {X 0,Y 344.924,Z 1260.924,A -85,B 0,C 180,E1 17467.161,E2 17467.161} C_VEL
LIN {X 0,Y 344.403,Z 1261.314,A -85,B 0,C 180,E1 17463.662,E2 17463.662} C_VEL
LIN {X 0,Y 344.207,Z 1260.063,A -85,B 0,C 180,E1 17460.333,E2 17460.333} C_VEL
LIN {X 0,Y 344.159,Z 1257.201,A -85,B 0,C 180,E1 17456.836,E2 17456.836} C_VEL
LIN {X 0,Y 344.292,Z 1252.904,A -85,B 0,C 180,E1 17453.496,E2 17453.496} C_VEL
LIN {X 0,Y 344.663,Z 1247.151,A -85,B 0,C 180,E1 17450.313,E2 17450.313} C_VEL
LIN {X 0,Y 345.471,Z 1239.397,A -85,B 0,C 180,E1 17446.953,E2 17446.953} C_VEL
LIN {X 0,Y 346.741,Z 1230.239,A -85,B 0,C 180,E1 17443.757,E2 17443.757} C_VEL
LIN {X 0,Y 348.611,Z 1219.037,A -85,B 0,C 180,E1 17440.566,E2 17440.566} C_VEL
LIN {X 0,Y 350.995,Z 1206.351,A -85,B 0,C 180,E1 17437.559,E2 17437.559} C_VEL
LIN {X 0,Y 353.859,Z 1192.151,A -85,B 0,C 180,E1 17434.721,E2 17434.721} C_VEL
LIN {X 0,Y 357.072,Z 1176.816,A -85,B 0,C 180,E1 17432.118,E2 17432.118} C_VEL
LIN {X 0,Y 360.72,Z 1159.358,A -85,B 0,C 180,E1 17429.61,E2 17429.61} C_VEL
LIN {X 0,Y 364.609,Z 1140.136,A -85,B 0,C 180,E1 17427.299,E2 17427.299} C_VEL
LIN {X 0,Y 368.323,Z 1120.73,A -85,B 0,C 180,E1 17425.344,E2 17425.344} C_VEL
LIN {X 0,Y 372.078,Z 1099.608,A -85,B 0,C 180,E1 17423.566,E2 17423.566} C_VEL
LIN {X 0,Y 375.67,Z 1076.982,A -85,B 0,C 180,E1 17422.008,E2 17422.008} C_VEL
LIN {X 0,Y 378.838,Z 1054.027,A -85,B 0,C 180,E1 17420.744,E2 17420.744} C_VEL
LIN {X 0,Y 381.488,Z 1030.92,A -85,B 0,C 180,E1 17419.753,E2 17419.753} C_VEL
LIN {X 0,Y 383.657,Z 1006.719,A -85,B 0,C 180,E1 17418.989,E2 17418.989} C_VEL
LIN {X 0,Y 400.368,Z 792.379,A -85,B 0,C 180,E1 17413.699,E2 17413.699} C_VEL
LIN {X 0,Y 385.335,Z 762.72,A -85,B 0,C 180,E1 17411.06,E2 17411.06} C_VEL
LIN {X 0,Y 370.36,Z 735.313,A -85,B 0,C 180,E1 17408.239,E2 17408.239} C_VEL
LIN {X 0,Y 357.085,Z 712.443,A -85,B 0,C 180,E1 17405.525,E2 17405.525} C_VEL
LIN {X 0,Y 350.112,Z 696.689,A -85,B 0,C 180,E1 17402.282,E2 17402.282} C_VEL
LIN {X 0,Y 347.122,Z 689.601,A -85,B 0,C 180,E1 17400.792,E2 17400.792} C_VEL
LIN {X 0,Y 347.088,Z 689.432,A -85,B 0,C 180,E1 17396.523,E2 17396.523} C_VEL
LIN {X 0,Y 347.09,Z 689.432,A -85,B 0,C 180,E1 17392.174,E2 17392.174} C_VEL
LIN {X 0,Y 347.095,Z 689.434,A -85,B 0,C 180,E1 17387.955,E2 17387.955} C_VEL
LIN {X 0,Y 347.089,Z 689.416,A -85,B 0,C 180,E1 17383.666,E2 17383.666} C_VEL
LIN {X 0,Y 347.086,Z 689.421,A -85,B 0,C 180,E1 17379.453,E2 17379.453} C_VEL
LIN {X 0,Y 347.088,Z 689.428,A -85,B 0,C 180,E1 17375.292,E2 17375.292} C_VEL
LIN {X 0,Y 347.09,Z 689.426,A -85,B 0,C 180,E1 17370.993,E2 17370.993} C_VEL
LIN {X 0,Y 347.084,Z 689.425,A -85,B 0,C 180,E1 17366.865,E2 17366.865} C_VEL
LIN {X 0,Y 347.089,Z 689.42,A -85,B 0,C 180,E1 17362.554,E2 17362.554} C_VEL
LIN {X 0,Y 347.091,Z 689.423,A -85,B 0,C 180,E1 17358.2,E2 17358.2} C_VEL
LIN {X 0,Y 347.087,Z 689.436,A -85,B 0,C 180,E1 17353.948,E2 17353.948} C_VEL
LIN {X 0,Y 347.112,Z 689.623,A -85,B 0,C 180,E1 17353.777,E2 17353.777} C_VEL
LIN {X 0,Y 348.479,Z 693.019,A -85,B 0,C 180,E1 17352.813,E2 17352.813} C_VEL
LIN {X 0,Y 349.383,Z 694.448,A -85,B 0,C 180,E1 17352.343,E2 17352.343} C_VEL
LIN {X 0,Y 354.101,Z 704.497,A -85,B 0,C 180,E1 17349.507,E2 17349.507} C_VEL
LIN {X 0,Y 359.358,Z 715.682,A -85,B 0,C 180,E1 17346.557,E2 17346.557} C_VEL
LIN {X 0,Y 365.597,Z 729.81,A -85,B 0,C 180,E1 17343.178,E2 17343.178} C_VEL
LIN {X 0,Y 372.161,Z 746.116,A -85,B 0,C 180,E1 17339.665,E2 17339.665} C_VEL
LIN {X 0,Y 378.499,Z 763.271,A -85,B 0,C 180,E1 17336.309,E2 17336.309} C_VEL
LIN {X 0,Y 384.884,Z 782.468,A -85,B 0,C 180,E1 17332.898,E2 17332.898} C_VEL
LIN {X 0,Y 387.932,Z 792.61,A -85,B 0,C 180,E1 17331.224,E2 17331.224} C_VEL
LIN {X 0,Y 380.409,Z 834.031,A -85,B 0,C 180,E1 17326.836,E2 17326.836} C_VEL
LIN {X 0,Y 373.319,Z 877.384,A -85,B 0,C 180,E1 17322.243,E2 17322.243} C_VEL
LIN {X 0,Y 367.15,Z 919.853,A -85,B 0,C 180,E1 17317.748,E2 17317.748} C_VEL
LIN {X 0,Y 366.375,Z 922.712,A -85,B 0,C 180,E1 17317.59,E2 17317.59} C_VEL
LIN {X 0,Y 360.622,Z 939.602,A -85,B 0,C 180,E1 17317.377,E2 17317.377} C_VEL
LIN {X 0,Y 358.913,Z 949.642,A -85,B 0,C 180,E1 17317.1,E2 17317.1} C_VEL
LIN {X 0,Y 358.484,Z 954.133,A -85,B 0,C 180,E1 17316.948,E2 17316.948} C_VEL
LIN {X 0,Y 352.878,Z 1026.073,A -85,B 0,C 180,E1 17314.379,E2 17314.379} C_VEL
LIN {X 0,Y 349.82,Z 1073.065,A -85,B 0,C 180,E1 17312.425,E2 17312.425} C_VEL
LIN {X 0,Y 348.648,Z 1089.827,A -85,B 0,C 180,E1 17311.464,E2 17311.464} C_VEL
LIN {X 0,Y 347.164,Z 1106.558,A -85,B 0,C 180,E1 17310.194,E2 17310.194} C_VEL
LIN {X 0,Y 345.484,Z 1122.483,A -85,B 0,C 180,E1 17308.633,E2 17308.633} C_VEL
LIN {X 0,Y 343.85,Z 1136.836,A -85,B 0,C 180,E1 17306.884,E2 17306.884} C_VEL
LIN {X 0,Y 342.11,Z 1151.234,A -85,B 0,C 180,E1 17304.705,E2 17304.705} C_VEL
LIN {X 0,Y 340.619,Z 1163.463,A -85,B 0,C 180,E1 17302.387,E2 17302.387} C_VEL
LIN {X 0,Y 339.468,Z 1173.807,A -85,B 0,C 180,E1 17299.979,E2 17299.979} C_VEL
LIN {X 0,Y 338.591,Z 1183.333,A -85,B 0,C 180,E1 17297.176,E2 17297.176} C_VEL
LIN {X 0,Y 338.182,Z 1190.239,A -85,B 0,C 180,E1 17294.556,E2 17294.556} C_VEL
LIN {X 0,Y 338.146,Z 1196.031,A -85,B 0,C 180,E1 17291.6,E2 17291.6} C_VEL
LIN {X 0,Y 338.536,Z 1199.804,A -85,B 0,C 180,E1 17288.664,E2 17288.664} C_VEL
LIN {X 0,Y 339.414,Z 1201.841,A -85,B 0,C 180,E1 17285.749,E2 17285.749} C_VEL
LIN {X 0,Y 340.95,Z 1202.027,A -85,B 0,C 180,E1 17282.689,E2 17282.689} C_VEL
LIN {X 0,Y 343.071,Z 1200.506,A -85,B 0,C 180,E1 17279.833,E2 17279.833} C_VEL
LIN {X 0,Y 346.071,Z 1197.019,A -85,B 0,C 180,E1 17276.853,E2 17276.853} C_VEL
LIN {X 0,Y 349.904,Z 1191.518,A -85,B 0,C 180,E1 17273.93,E2 17273.93} C_VEL
LIN {X 0,Y 354.026,Z 1184.879,A -85,B 0,C 180,E1 17271.391,E2 17271.391} C_VEL
LIN {X 0,Y 359.113,Z 1175.748,A -85,B 0,C 180,E1 17268.761,E2 17268.761} C_VEL
LIN {X 0,Y 364.595,Z 1164.902,A -85,B 0,C 180,E1 17266.358,E2 17266.358} C_VEL
LIN {X 0,Y 370.723,Z 1151.438,A -85,B 0,C 180,E1 17264.031,E2 17264.031} C_VEL
LIN {X 0,Y 376.676,Z 1136.85,A -85,B 0,C 180,E1 17262.066,E2 17262.066} C_VEL
LIN {X 0,Y 382.228,Z 1121.578,A -85,B 0,C 180,E1 17260.437,E2 17260.437} C_VEL
LIN {X 0,Y 387.446,Z 1105.28,A -85,B 0,C 180,E1 17259.057,E2 17259.057} C_VEL
LIN {X 0,Y 394.999,Z 1079.502,A -85,B 0,C 180,E1 17257.37,E2 17257.37} C_VEL
LIN {X 0,Y 404.222,Z 1048.946,A -85,B 0,C 180,E1 17255.756,E2 17255.756} C_VEL
LIN {X 0,Y 413.995,Z 1013.876,A -85,B 0,C 180,E1 17254.231,E2 17254.231} C_VEL
LIN {X 0,Y 422.02,Z 979.76,A -85,B 0,C 180,E1 17252.989,E2 17252.989} C_VEL
LIN {X 0,Y 424.264,Z 968.936,A -85,B 0,C 180,E1 17252.603,E2 17252.603} C_VEL
LIN {X 0,Y 425.582,Z 957.296,A -85,B 0,C 180,E1 17251.514,E2 17251.514} C_VEL
LIN {X 0,Y 442.441,Z 929.527,A -85,B 0,C 180,E1 17247.921,E2 17247.921} C_VEL
LIN {X 0,Y 446.149,Z 924.002,A -85,B 0,C 180,E1 17247.181,E2 17247.181} C_VEL
LIN {X 0,Y 436.162,Z 940.933,A -85,B 0,C 180,E1 17244.694,E2 17244.694} C_VEL
LIN {X 0,Y 428.759,Z 957.611,A -85,B 0,C 180,E1 17242,E2 17242} C_VEL
LIN {X 0,Y 424.401,Z 973.045,A -85,B 0,C 180,E1 17239.34,E2 17239.34} C_VEL
LIN {X 0,Y 423.994,Z 976.75,A -85,B 0,C 180,E1 17238.721,E2 17238.721} C_VEL
LIN {X 0,Y 424.241,Z 980.019,A -85,B 0,C 180,E1 17238.294,E2 17238.294} C_VEL
LIN {X 0,Y 420.548,Z 999.544,A -85,B 0,C 180,E1 17237.888,E2 17237.888} C_VEL
LIN {X 0,Y 415.012,Z 1024.402,A -85,B 0,C 180,E1 17237.443,E2 17237.443} C_VEL
LIN {X 0,Y 410,Z 1045.082,A -85,B 0,C 180,E1 17236.815,E2 17236.815} C_VEL
LIN {X 0,Y 403.609,Z 1068.761,A -85,B 0,C 180,E1 17235.82,E2 17235.82} C_VEL
LIN {X 0,Y 396.245,Z 1092.995,A -85,B 0,C 180,E1 17234.544,E2 17234.544} C_VEL
LIN {X 0,Y 388.294,Z 1116.918,A -85,B 0,C 180,E1 17232.927,E2 17232.927} C_VEL
LIN {X 0,Y 380.778,Z 1138.314,A -85,B 0,C 180,E1 17231.128,E2 17231.128} C_VEL
LIN {X 0,Y 373.435,Z 1158.26,A -85,B 0,C 180,E1 17229.088,E2 17229.088} C_VEL
LIN {X 0,Y 365.967,Z 1177.77,A -85,B 0,C 180,E1 17226.651,E2 17226.651} C_VEL
LIN {X 0,Y 359.208,Z 1195.118,A -85,B 0,C 180,E1 17224.018,E2 17224.018} C_VEL
LIN {X 0,Y 353.242,Z 1210.604,A -85,B 0,C 180,E1 17221.195,E2 17221.195} C_VEL
LIN {X 0,Y 348.017,Z 1224.767,A -85,B 0,C 180,E1 17218.108,E2 17218.108} C_VEL
LIN {X 0,Y 343.671,Z 1237.506,A -85,B 0,C 180,E1 17214.766,E2 17214.766} C_VEL
LIN {X 0,Y 340.228,Z 1249.166,A -85,B 0,C 180,E1 17211.008,E2 17211.008} C_VEL
LIN {X 0,Y 338.554,Z 1256.457,A -85,B 0,C 180,E1 17208.241,E2 17208.241} C_VEL
LIN {X 0,Y 337.327,Z 1266.226,A -85,B 0,C 180,E1 17205.118,E2 17205.118} C_VEL
LIN {X 0,Y 336.621,Z 1274.687,A -85,B 0,C 180,E1 17201.824,E2 17201.824} C_VEL
LIN {X 0,Y 336.385,Z 1280.984,A -85,B 0,C 180,E1 17198.717,E2 17198.717} C_VEL
LIN {X 0,Y 336.407,Z 1285.923,A -85,B 0,C 180,E1 17195.455,E2 17195.455} C_VEL
LIN {X 0,Y 336.47,Z 1289.14,A -85,B 0,C 180,E1 17192.382,E2 17192.382} C_VEL
LIN {X 0,Y 336.434,Z 1290.915,A -85,B 0,C 180,E1 17189.146,E2 17189.146} C_VEL
LIN {X 0,Y 336.25,Z 1291.279,A -85,B 0,C 180,E1 17185.905,E2 17185.905} C_VEL
LIN {X 0,Y 336.157,Z 1289.971,A -85,B 0,C 180,E1 17182.478,E2 17182.478} C_VEL
LIN {X 0,Y 336.434,Z 1287.032,A -85,B 0,C 180,E1 17178.859,E2 17178.859} C_VEL
LIN {X 0,Y 337.457,Z 1282.391,A -85,B 0,C 180,E1 17175.235,E2 17175.235} C_VEL
LIN {X 0,Y 339.528,Z 1275.731,A -85,B 0,C 180,E1 17171.453,E2 17171.453} C_VEL
LIN {X 0,Y 342.804,Z 1267.265,A -85,B 0,C 180,E1 17167.715,E2 17167.715} C_VEL
LIN {X 0,Y 347.42,Z 1256.93,A -85,B 0,C 180,E1 17164.056,E2 17164.056} C_VEL
LIN {X 0,Y 353.748,Z 1243.97,A -85,B 0,C 180,E1 17160.351,E2 17160.351} C_VEL
LIN {X 0,Y 361.321,Z 1229.51,A -85,B 0,C 180,E1 17156.962,E2 17156.962} C_VEL
LIN {X 0,Y 370.429,Z 1213.015,A -85,B 0,C 180,E1 17153.76,E2 17153.76} C_VEL
LIN {X 0,Y 381.135,Z 1194.425,A -85,B 0,C 180,E1 17150.782,E2 17150.782} C_VEL
LIN {X 0,Y 393.229,Z 1174.135,A -85,B 0,C 180,E1 17148.126,E2 17148.126} C_VEL
LIN {X 0,Y 405.664,Z 1153.796,A -85,B 0,C 180,E1 17145.965,E2 17145.965} C_VEL
LIN {X 0,Y 418.429,Z 1133.067,A -85,B 0,C 180,E1 17144.2,E2 17144.2} C_VEL
LIN {X 0,Y 405.492,Z 1153.224,A -85,B 0,C 180,E1 17142.123,E2 17142.123} C_VEL
LIN {X 0,Y 393.123,Z 1172.316,A -85,B 0,C 180,E1 17139.673,E2 17139.673} C_VEL
LIN {X 0,Y 381.648,Z 1190.025,A -85,B 0,C 180,E1 17136.868,E2 17136.868} C_VEL
LIN {X 0,Y 371.62,Z 1205.589,A -85,B 0,C 180,E1 17133.846,E2 17133.846} C_VEL
LIN {X 0,Y 362.994,Z 1219.106,A -85,B 0,C 180,E1 17130.637,E2 17130.637} C_VEL
LIN {X 0,Y 355.394,Z 1231.085,A -85,B 0,C 180,E1 17127.115,E2 17127.115} C_VEL
LIN {X 0,Y 349.215,Z 1240.985,A -85,B 0,C 180,E1 17123.453,E2 17123.453} C_VEL
LIN {X 0,Y 344.588,Z 1248.59,A -85,B 0,C 180,E1 17119.846,E2 17119.846} C_VEL
LIN {X 0,Y 341.014,Z 1254.677,A -85,B 0,C 180,E1 17115.999,E2 17115.999} C_VEL
LIN {X 0,Y 338.679,Z 1258.794,A -85,B 0,C 180,E1 17112.247,E2 17112.247} C_VEL
LIN {X 0,Y 337.279,Z 1261.177,A -85,B 0,C 180,E1 17108.524,E2 17108.524} C_VEL
LIN {X 0,Y 336.559,Z 1261.802,A -85,B 0,C 180,E1 17104.943,E2 17104.943} C_VEL
LIN {X 0,Y 336.252,Z 1260.893,A -85,B 0,C 180,E1 17101.363,E2 17101.363} C_VEL
LIN {X 0,Y 336.165,Z 1258.805,A -85,B 0,C 180,E1 17098.296,E2 17098.296} C_VEL
LIN {X 0,Y 336.212,Z 1254.996,A -85,B 0,C 180,E1 17094.881,E2 17094.881} C_VEL
LIN {X 0,Y 336.475,Z 1249.932,A -85,B 0,C 180,E1 17091.627,E2 17091.627} C_VEL
LIN {X 0,Y 337.11,Z 1242.754,A -85,B 0,C 180,E1 17088.188,E2 17088.188} C_VEL
LIN {X 0,Y 338.193,Z 1234.207,A -85,B 0,C 180,E1 17084.919,E2 17084.919} C_VEL
LIN {X 0,Y 339.866,Z 1223.795,A -85,B 0,C 180,E1 17081.651,E2 17081.651} C_VEL
LIN {X 0,Y 342.063,Z 1211.966,A -85,B 0,C 180,E1 17078.568,E2 17078.568} C_VEL
LIN {X 0,Y 344.815,Z 1198.237,A -85,B 0,C 180,E1 17075.582,E2 17075.582} C_VEL
LIN {X 0,Y 348.092,Z 1182.694,A -85,B 0,C 180,E1 17072.731,E2 17072.731} C_VEL
LIN {X 0,Y 351.893,Z 1164.931,A -85,B 0,C 180,E1 17069.993,E2 17069.993} C_VEL
LIN {X 0,Y 355.735,Z 1146.643,A -85,B 0,C 180,E1 17067.625,E2 17067.625} C_VEL
LIN {X 0,Y 359.583,Z 1127.519,A -85,B 0,C 180,E1 17065.537,E2 17065.537} C_VEL
LIN {X 0,Y 363.467,Z 1106.737,A -85,B 0,C 180,E1 17063.641,E2 17063.641} C_VEL
LIN {X 0,Y 367.164,Z 1084.977,A -85,B 0,C 180,E1 17062.014,E2 17062.014} C_VEL
LIN {X 0,Y 370.517,Z 1062.316,A -85,B 0,C 180,E1 17060.641,E2 17060.641} C_VEL
LIN {X 0,Y 373.423,Z 1039.149,A -85,B 0,C 180,E1 17059.534,E2 17059.534} C_VEL
LIN {X 0,Y 375.906,Z 1014.705,A -85,B 0,C 180,E1 17058.661,E2 17058.661} C_VEL
LIN {X 0,Y 393.617,Z 794.934,A -85,B 0,C 180,E1 17053.081,E2 17053.081} C_VEL
LIN {X 0,Y 378.972,Z 766.084,A -85,B 0,C 180,E1 17050.447,E2 17050.447} C_VEL
LIN {X 0,Y 364.775,Z 739.977,A -85,B 0,C 180,E1 17047.708,E2 17047.708} C_VEL
LIN {X 0,Y 350.804,Z 716.058,A -85,B 0,C 180,E1 17044.806,E2 17044.806} C_VEL
LIN {X 0,Y 348.966,Z 712.776,A -85,B 0,C 180,E1 17044.367,E2 17044.367} C_VEL
LIN {X 0,Y 342.181,Z 697.647,A -85,B 0,C 180,E1 17041.148,E2 17041.148} C_VEL
LIN {X 0,Y 340.116,Z 693.326,A -85,B 0,C 180,E1 17040.182,E2 17040.182} C_VEL
LIN {X 0,Y 339.15,Z 690.415,A -85,B 0,C 180,E1 17039.573,E2 17039.573} C_VEL
LIN {X 0,Y 339.158,Z 690.424,A -85,B 0,C 180,E1 17035.165,E2 17035.165} C_VEL
LIN {X 0,Y 339.157,Z 690.422,A -85,B 0,C 180,E1 17030.841,E2 17030.841} C_VEL
LIN {X 0,Y 339.15,Z 690.418,A -85,B 0,C 180,E1 17026.619,E2 17026.619} C_VEL
LIN {X 0,Y 339.152,Z 690.404,A -85,B 0,C 180,E1 17022.43,E2 17022.43} C_VEL
LIN {X 0,Y 339.156,Z 690.402,A -85,B 0,C 180,E1 17018.138,E2 17018.138} C_VEL
LIN {X 0,Y 339.145,Z 690.406,A -85,B 0,C 180,E1 17013.89,E2 17013.89} C_VEL
LIN {X 0,Y 339.148,Z 690.406,A -85,B 0,C 180,E1 17009.664,E2 17009.664} C_VEL
LIN {X 0,Y 339.155,Z 690.409,A -85,B 0,C 180,E1 17005.267,E2 17005.267} C_VEL
LIN {X 0,Y 339.148,Z 690.418,A -85,B 0,C 180,E1 17000.993,E2 17000.993} C_VEL
LIN {X 0,Y 339.152,Z 690.418,A -85,B 0,C 180,E1 16996.634,E2 16996.634} C_VEL
LIN {X 0,Y 339.192,Z 690.609,A -85,B 0,C 180,E1 16995.492,E2 16995.492} C_VEL
LIN {X 0,Y 340.495,Z 693.956,A -85,B 0,C 180,E1 16994.503,E2 16994.503} C_VEL
LIN {X 0,Y 341.628,Z 695.875,A -85,B 0,C 180,E1 16993.859,E2 16993.859} C_VEL
LIN {X 0,Y 344.149,Z 701.218,A -85,B 0,C 180,E1 16992.24,E2 16992.24} C_VEL
LIN {X 0,Y 347.927,Z 708.857,A -85,B 0,C 180,E1 16990.005,E2 16990.005} C_VEL
LIN {X 0,Y 353.647,Z 721.343,A -85,B 0,C 180,E1 16986.685,E2 16986.685} C_VEL
LIN {X 0,Y 359.562,Z 734.872,A -85,B 0,C 180,E1 16983.406,E2 16983.406} C_VEL
LIN {X 0,Y 366.069,Z 751.258,A -85,B 0,C 180,E1 16979.832,E2 16979.832} C_VEL
LIN {X 0,Y 372.336,Z 768.534,A -85,B 0,C 180,E1 16976.416,E2 16976.416} C_VEL
LIN {X 0,Y 378.324,Z 786.771,A -85,B 0,C 180,E1 16973.137,E2 16973.137} C_VEL
LIN {X 0,Y 380.909,Z 795.495,A -85,B 0,C 180,E1 16971.674,E2 16971.674} C_VEL
LIN {X 0,Y 373.047,Z 837.61,A -85,B 0,C 180,E1 16967.157,E2 16967.157} C_VEL
LIN {X 0,Y 365.62,Z 881.802,A -85,B 0,C 180,E1 16962.41,E2 16962.41} C_VEL
LIN {X 0,Y 359.647,Z 922.686,A -85,B 0,C 180,E1 16958.06,E2 16958.06} C_VEL
LIN {X 0,Y 359.979,Z 934.905,A -85,B 0,C 180,E1 16957.574,E2 16957.574} C_VEL
LIN {X 0,Y 358.484,Z 954.133,A -85,B 0,C 180,E1 16956.948,E2 16956.948} C_VEL
LIN {X 0,Y 356.948,Z 961.658,A -85,B 0,C 180,E1 16956.762,E2 16956.762} C_VEL
LIN {X 0,Y 349.61,Z 981.503,A -85,B 0,C 180,E1 16956.453,E2 16956.453} C_VEL
LIN {X 0,Y 348.394,Z 987.945,A -85,B 0,C 180,E1 16956.262,E2 16956.262} C_VEL
LIN {X 0,Y 343.199,Z 1054.694,A -85,B 0,C 180,E1 16953.618,E2 16953.618} C_VEL
LIN {X 0,Y 341.71,Z 1079.674,A -85,B 0,C 180,E1 16952.445,E2 16952.445} C_VEL
LIN {X 0,Y 340.358,Z 1096.745,A -85,B 0,C 180,E1 16951.331,E2 16951.331} C_VEL
LIN {X 0,Y 338.736,Z 1113.209,A -85,B 0,C 180,E1 16949.925,E2 16949.925} C_VEL
LIN {X 0,Y 337.102,Z 1127.865,A -85,B 0,C 180,E1 16948.332,E2 16948.332} C_VEL
LIN {X 0,Y 335.341,Z 1142.438,A -85,B 0,C 180,E1 16946.377,E2 16946.377} C_VEL
LIN {X 0,Y 333.614,Z 1156.311,A -85,B 0,C 180,E1 16944.055,E2 16944.055} C_VEL
LIN {X 0,Y 332.242,Z 1167.595,A -85,B 0,C 180,E1 16941.726,E2 16941.726} C_VEL
LIN {X 0,Y 331.121,Z 1178.139,A -85,B 0,C 180,E1 16939.034,E2 16939.034} C_VEL
LIN {X 0,Y 330.404,Z 1186.909,A -85,B 0,C 180,E1 16936.166,E2 16936.166} C_VEL
LIN {X 0,Y 330.142,Z 1193.225,A -85,B 0,C 180,E1 16933.486,E2 16933.486} C_VEL
LIN {X 0,Y 330.293,Z 1198.626,A -85,B 0,C 180,E1 16930.289,E2 16930.289} C_VEL
LIN {X 0,Y 330.919,Z 1201.8,A -85,B 0,C 180,E1 16927.291,E2 16927.291} C_VEL
LIN {X 0,Y 332.185,Z 1203.277,A -85,B 0,C 180,E1 16924.143,E2 16924.143} C_VEL
LIN {X 0,Y 334.276,Z 1202.717,A -85,B 0,C 180,E1 16920.857,E2 16920.857} C_VEL
LIN {X 0,Y 336.901,Z 1200.428,A -85,B 0,C 180,E1 16917.959,E2 16917.959} C_VEL
LIN {X 0,Y 340.506,Z 1196.208,A -85,B 0,C 180,E1 16914.946,E2 16914.946} C_VEL
LIN {X 0,Y 344.968,Z 1189.895,A -85,B 0,C 180,E1 16912.003,E2 16912.003} C_VEL
LIN {X 0,Y 349.975,Z 1181.942,A -85,B 0,C 180,E1 16909.298,E2 16909.298} C_VEL
LIN {X 0,Y 355.129,Z 1172.912,A -85,B 0,C 180,E1 16906.94,E2 16906.94} C_VEL
LIN {X 0,Y 361.101,Z 1161.448,A -85,B 0,C 180,E1 16904.584,E2 16904.584} C_VEL
LIN {X 0,Y 367.397,Z 1147.993,A -85,B 0,C 180,E1 16902.417,E2 16902.417} C_VEL
LIN {X 0,Y 373.627,Z 1133.134,A -85,B 0,C 180,E1 16900.538,E2 16900.538} C_VEL
LIN {X 0,Y 379.373,Z 1117.797,A -85,B 0,C 180,E1 16898.995,E2 16898.995} C_VEL
LIN {X 0,Y 384.999,Z 1100.646,A -85,B 0,C 180,E1 16897.637,E2 16897.637} C_VEL
LIN {X 0,Y 393.922,Z 1072.596,A -85,B 0,C 180,E1 16895.879,E2 16895.879} C_VEL
LIN {X 0,Y 403.896,Z 1041.038,A -85,B 0,C 180,E1 16894.3,E2 16894.3} C_VEL
LIN {X 0,Y 413.278,Z 1007.715,A -85,B 0,C 180,E1 16892.91,E2 16892.91} C_VEL
LIN {X 0,Y 421.001,Z 974.74,A -85,B 0,C 180,E1 16891.76,E2 16891.76} C_VEL
LIN {X 0,Y 421.637,Z 971.485,A -85,B 0,C 180,E1 16891.613,E2 16891.613} C_VEL
LIN {X 0,Y 423.37,Z 959.129,A -85,B 0,C 180,E1 16890.422,E2 16890.422} C_VEL
LIN {X 0,Y 439.387,Z 933.983,A -85,B 0,C 180,E1 16887.153,E2 16887.153} C_VEL
LIN {X 0,Y 429.575,Z 950.88,A -85,B 0,C 180,E1 16884.55,E2 16884.55} C_VEL
LIN {X 0,Y 422.587,Z 967.435,A -85,B 0,C 180,E1 16881.767,E2 16881.767} C_VEL
LIN {X 0,Y 420.798,Z 973.813,A -85,B 0,C 180,E1 16880.665,E2 16880.665} C_VEL
LIN {X 0,Y 421.154,Z 983.609,A -85,B 0,C 180,E1 16879.249,E2 16879.249} C_VEL
LIN {X 0,Y 417.721,Z 1000.689,A -85,B 0,C 180,E1 16878.909,E2 16878.909} C_VEL
LIN {X 0,Y 411.502,Z 1027.249,A -85,B 0,C 180,E1 16878.415,E2 16878.415} C_VEL
LIN {X 0,Y 406.35,Z 1047.115,A -85,B 0,C 180,E1 16877.784,E2 16877.784} C_VEL
LIN {X 0,Y 398.072,Z 1075.477,A -85,B 0,C 180,E1 16876.541,E2 16876.541} C_VEL
LIN {X 0,Y 389.986,Z 1099.847,A -85,B 0,C 180,E1 16875.154,E2 16875.154} C_VEL
LIN {X 0,Y 382.203,Z 1121.796,A -85,B 0,C 180,E1 16873.575,E2 16873.575} C_VEL
LIN {X 0,Y 373.508,Z 1144.862,A -85,B 0,C 180,E1 16871.513,E2 16871.513} C_VEL
LIN {X 0,Y 365.763,Z 1164.324,A -85,B 0,C 180,E1 16869.359,E2 16869.359} C_VEL
LIN {X 0,Y 358.388,Z 1182.17,A -85,B 0,C 180,E1 16866.955,E2 16866.955} C_VEL
LIN {X 0,Y 351.502,Z 1198.684,A -85,B 0,C 180,E1 16864.277,E2 16864.277} C_VEL
LIN {X 0,Y 345.254,Z 1213.879,A -85,B 0,C 180,E1 16861.312,E2 16861.312} C_VEL
LIN {X 0,Y 339.581,Z 1228.279,A -85,B 0,C 180,E1 16857.913,E2 16857.913} C_VEL
LIN {X 0,Y 335.101,Z 1240.766,A -85,B 0,C 180,E1 16854.313,E2 16854.313} C_VEL
LIN {X 0,Y 331.746,Z 1251.745,A -85,B 0,C 180,E1 16850.386,E2 16850.386} C_VEL
LIN {X 0,Y 330.258,Z 1258.367,A -85,B 0,C 180,E1 16847.621,E2 16847.621} C_VEL
LIN {X 0,Y 329.09,Z 1268.319,A -85,B 0,C 180,E1 16844.245,E2 16844.245} C_VEL
LIN {X 0,Y 328.542,Z 1275.81,A -85,B 0,C 180,E1 16841.051,E2 16841.051} C_VEL
LIN {X 0,Y 328.397,Z 1282.042,A -85,B 0,C 180,E1 16837.697,E2 16837.697} C_VEL
LIN {X 0,Y 328.452,Z 1286.133,A -85,B 0,C 180,E1 16834.712,E2 16834.712} C_VEL
LIN {X 0,Y 328.505,Z 1289.183,A -85,B 0,C 180,E1 16831.393,E2 16831.393} C_VEL
LIN {X 0,Y 328.418,Z 1290.551,A -85,B 0,C 180,E1 16828.427,E2 16828.427} C_VEL
LIN {X 0,Y 328.211,Z 1290.699,A -85,B 0,C 180,E1 16825.008,E2 16825.008} C_VEL
LIN {X 0,Y 328.174,Z 1289.273,A -85,B 0,C 180,E1 16821.588,E2 16821.588} C_VEL
LIN {X 0,Y 328.665,Z 1285.96,A -85,B 0,C 180,E1 16817.702,E2 16817.702} C_VEL
LIN {X 0,Y 330.085,Z 1280.916,A -85,B 0,C 180,E1 16813.816,E2 16813.816} C_VEL
LIN {X 0,Y 332.654,Z 1273.989,A -85,B 0,C 180,E1 16809.959,E2 16809.959} C_VEL
LIN {X 0,Y 336.518,Z 1265.262,A -85,B 0,C 180,E1 16806.164,E2 16806.164} C_VEL
LIN {X 0,Y 341.952,Z 1254.453,A -85,B 0,C 180,E1 16802.374,E2 16802.374} C_VEL
LIN {X 0,Y 348.926,Z 1241.787,A -85,B 0,C 180,E1 16798.754,E2 16798.754} C_VEL
LIN {X 0,Y 357.694,Z 1226.692,A -85,B 0,C 180,E1 16795.23,E2 16795.23} C_VEL
LIN {X 0,Y 367.724,Z 1210.263,A -85,B 0,C 180,E1 16792.081,E2 16792.081} C_VEL
LIN {X 0,Y 379.363,Z 1191.933,A -85,B 0,C 180,E1 16789.18,E2 16789.18} C_VEL
LIN {X 0,Y 392.083,Z 1172.59,A -85,B 0,C 180,E1 16786.684,E2 16786.684} C_VEL
LIN {X 0,Y 405.336,Z 1152.858,A -85,B 0,C 180,E1 16784.627,E2 16784.627} C_VEL
LIN {X 0,Y 409.119,Z 1147.229,A -85,B 0,C 180,E1 16784.102,E2 16784.102} C_VEL
LIN {X 0,Y 395.624,Z 1166.277,A -85,B 0,C 180,E1 16781.854,E2 16781.854} C_VEL
LIN {X 0,Y 382.824,Z 1184.286,A -85,B 0,C 180,E1 16779.204,E2 16779.204} C_VEL
LIN {X 0,Y 371.515,Z 1200.275,A -85,B 0,C 180,E1 16776.307,E2 16776.307} C_VEL
LIN {X 0,Y 361.249,Z 1214.891,A -85,B 0,C 180,E1 16773.043,E2 16773.043} C_VEL
LIN {X 0,Y 352.858,Z 1226.965,A -85,B 0,C 180,E1 16769.729,E2 16769.729} C_VEL
LIN {X 0,Y 345.542,Z 1237.611,A -85,B 0,C 180,E1 16766.094,E2 16766.094} C_VEL
LIN {X 0,Y 339.447,Z 1246.619,A -85,B 0,C 180,E1 16762.151,E2 16762.151} C_VEL
LIN {X 0,Y 335.011,Z 1253.28,A -85,B 0,C 180,E1 16758.264,E2 16758.264} C_VEL
LIN {X 0,Y 331.985,Z 1257.916,A -85,B 0,C 180,E1 16754.477,E2 16754.477} C_VEL
LIN {X 0,Y 330.003,Z 1260.934,A -85,B 0,C 180,E1 16750.651,E2 16750.651} C_VEL
LIN {X 0,Y 328.928,Z 1262.256,A -85,B 0,C 180,E1 16746.984,E2 16746.984} C_VEL
LIN {X 0,Y 328.384,Z 1261.945,A -85,B 0,C 180,E1 16743.317,E2 16743.317} C_VEL
LIN {X 0,Y 328.206,Z 1260.087,A -85,B 0,C 180,E1 16739.651,E2 16739.651} C_VEL
LIN {X 0,Y 328.166,Z 1256.963,A -85,B 0,C 180,E1 16736.331,E2 16736.331} C_VEL
LIN {X 0,Y 328.35,Z 1252.067,A -85,B 0,C 180,E1 16732.828,E2 16732.828} C_VEL
LIN {X 0,Y 328.85,Z 1245.502,A -85,B 0,C 180,E1 16729.311,E2 16729.311} C_VEL
LIN {X 0,Y 329.783,Z 1237.529,A -85,B 0,C 180,E1 16725.962,E2 16725.962} C_VEL
LIN {X 0,Y 331.276,Z 1227.645,A -85,B 0,C 180,E1 16722.614,E2 16722.614} C_VEL
LIN {X 0,Y 333.431,Z 1215.737,A -85,B 0,C 180,E1 16719.276,E2 16719.276} C_VEL
LIN {X 0,Y 335.979,Z 1203.139,A -85,B 0,C 180,E1 16716.311,E2 16716.311} C_VEL
LIN {X 0,Y 339.147,Z 1188.342,A -85,B 0,C 180,E1 16713.376,E2 16713.376} C_VEL
LIN {X 0,Y 342.706,Z 1171.984,A -85,B 0,C 180,E1 16710.649,E2 16710.649} C_VEL
LIN {X 0,Y 346.446,Z 1154.75,A -85,B 0,C 180,E1 16708.216,E2 16708.216} C_VEL
LIN {X 0,Y 350.663,Z 1134.599,A -85,B 0,C 180,E1 16705.824,E2 16705.824} C_VEL
LIN {X 0,Y 354.648,Z 1114.326,A -85,B 0,C 180,E1 16703.818,E2 16703.818} C_VEL
LIN {X 0,Y 358.55,Z 1092.799,A -85,B 0,C 180,E1 16702.054,E2 16702.054} C_VEL
LIN {X 0,Y 362.121,Z 1070.68,A -85,B 0,C 180,E1 16700.574,E2 16700.574} C_VEL
LIN {X 0,Y 365.379,Z 1046.9,A -85,B 0,C 180,E1 16699.312,E2 16699.312} C_VEL
LIN {X 0,Y 368.133,Z 1022.156,A -85,B 0,C 180,E1 16698.321,E2 16698.321} C_VEL
LIN {X 0,Y 370.962,Z 987.819,A -85,B 0,C 180,E1 16697.353,E2 16697.353} C_VEL
LIN {X 0,Y 386.985,Z 797.749,A -85,B 0,C 180,E1 16692.467,E2 16692.467} C_VEL
LIN {X 0,Y 372.254,Z 768.644,A -85,B 0,C 180,E1 16689.74,E2 16689.74} C_VEL
LIN {X 0,Y 357.528,Z 741.618,A -85,B 0,C 180,E1 16686.814,E2 16686.814} C_VEL
LIN {X 0,Y 343.435,Z 717.579,A -85,B 0,C 180,E1 16683.787,E2 16683.787} C_VEL
LIN {X 0,Y 340.676,Z 712.811,A -85,B 0,C 180,E1 16683.089,E2 16683.089} C_VEL
LIN {X 0,Y 334.262,Z 698.638,A -85,B 0,C 180,E1 16679.973,E2 16679.973} C_VEL
LIN {X 0,Y 332.22,Z 694.406,A -85,B 0,C 180,E1 16678.986,E2 16678.986} C_VEL
LIN {X 0,Y 331.221,Z 691.407,A -85,B 0,C 180,E1 16678.293,E2 16678.293} C_VEL
LIN {X 0,Y 331.22,Z 691.408,A -85,B 0,C 180,E1 16673.836,E2 16673.836} C_VEL
LIN {X 0,Y 331.211,Z 691.406,A -85,B 0,C 180,E1 16669.397,E2 16669.397} C_VEL
LIN {X 0,Y 331.213,Z 691.409,A -85,B 0,C 180,E1 16664.973,E2 16664.973} C_VEL
LIN {X 0,Y 331.216,Z 691.411,A -85,B 0,C 180,E1 16660.614,E2 16660.614} C_VEL
LIN {X 0,Y 331.22,Z 691.411,A -85,B 0,C 180,E1 16656.241,E2 16656.241} C_VEL
LIN {X 0,Y 331.208,Z 691.413,A -85,B 0,C 180,E1 16651.732,E2 16651.732} C_VEL
LIN {X 0,Y 331.207,Z 691.41,A -85,B 0,C 180,E1 16647.407,E2 16647.407} C_VEL
LIN {X 0,Y 331.212,Z 691.401,A -85,B 0,C 180,E1 16643.067,E2 16643.067} C_VEL
LIN {X 0,Y 331.208,Z 691.399,A -85,B 0,C 180,E1 16638.686,E2 16638.686} C_VEL
LIN {X 0,Y 331.224,Z 691.504,A -85,B 0,C 180,E1 16637.36,E2 16637.36} C_VEL
LIN {X 0,Y 332.608,Z 695.005,A -85,B 0,C 180,E1 16636.264,E2 16636.264} C_VEL
LIN {X 0,Y 333.713,Z 696.804,A -85,B 0,C 180,E1 16635.603,E2 16635.603} C_VEL
LIN {X 0,Y 336.421,Z 702.535,A -85,B 0,C 180,E1 16633.779,E2 16633.779} C_VEL
LIN {X 0,Y 338.754,Z 707.294,A -85,B 0,C 180,E1 16632.303,E2 16632.303} C_VEL
LIN {X 0,Y 343.771,Z 717.546,A -85,B 0,C 180,E1 16629.308,E2 16629.308} C_VEL
LIN {X 0,Y 350.453,Z 732.608,A -85,B 0,C 180,E1 16625.385,E2 16625.385} C_VEL
LIN {X 0,Y 357.168,Z 749.013,A -85,B 0,C 180,E1 16621.584,E2 16621.584} C_VEL
LIN {X 0,Y 363.657,Z 766.452,A -85,B 0,C 180,E1 16617.953,E2 16617.953} C_VEL
LIN {X 0,Y 369.579,Z 784.048,A -85,B 0,C 180,E1 16614.625,E2 16614.625} C_VEL
LIN {X 0,Y 373.911,Z 798.314,A -85,B 0,C 180,E1 16612.145,E2 16612.145} C_VEL
LIN {X 0,Y 365.654,Z 841.312,A -85,B 0,C 180,E1 16607.473,E2 16607.473} C_VEL
LIN {X 0,Y 357.979,Z 885.732,A -85,B 0,C 180,E1 16602.636,E2 16602.636} C_VEL
LIN {X 0,Y 352.314,Z 923.382,A -85,B 0,C 180,E1 16598.566,E2 16598.566} C_VEL
LIN {X 0,Y 352.615,Z 935.64,A -85,B 0,C 180,E1 16598.073,E2 16598.073} C_VEL
LIN {X 0,Y 348.394,Z 987.945,A -85,B 0,C 180,E1 16596.262,E2 16596.262} C_VEL
LIN {X 0,Y 346.838,Z 995.436,A -85,B 0,C 180,E1 16596.044,E2 16596.044} C_VEL
LIN {X 0,Y 339.368,Z 1015.179,A -85,B 0,C 180,E1 16595.643,E2 16595.643} C_VEL
LIN {X 0,Y 338.128,Z 1021.601,A -85,B 0,C 180,E1 16595.428,E2 16595.428} C_VEL
LIN {X 0,Y 334.572,Z 1071.178,A -85,B 0,C 180,E1 16593.27,E2 16593.27} C_VEL
LIN {X 0,Y 333.339,Z 1088.656,A -85,B 0,C 180,E1 16592.272,E2 16592.272} C_VEL
LIN {X 0,Y 331.838,Z 1104.968,A -85,B 0,C 180,E1 16591.015,E2 16591.015} C_VEL
LIN {X 0,Y 330.044,Z 1121.428,A -85,B 0,C 180,E1 16589.393,E2 16589.393} C_VEL
LIN {X 0,Y 328.143,Z 1137.388,A -85,B 0,C 180,E1 16587.395,E2 16587.395} C_VEL
LIN {X 0,Y 326.435,Z 1150.865,A -85,B 0,C 180,E1 16585.296,E2 16585.296} C_VEL
LIN {X 0,Y 324.917,Z 1162.937,A -85,B 0,C 180,E1 16583.006,E2 16583.006} C_VEL
LIN {X 0,Y 323.639,Z 1173.889,A -85,B 0,C 180,E1 16580.433,E2 16580.433} C_VEL
LIN {X 0,Y 322.776,Z 1182.74,A -85,B 0,C 180,E1 16577.859,E2 16577.859} C_VEL
LIN {X 0,Y 322.252,Z 1190.641,A -85,B 0,C 180,E1 16574.924,E2 16574.924} C_VEL
LIN {X 0,Y 322.172,Z 1196.617,A -85,B 0,C 180,E1 16572.002,E2 16572.002} C_VEL
LIN {X 0,Y 322.588,Z 1201.23,A -85,B 0,C 180,E1 16568.736,E2 16568.736} C_VEL
LIN {X 0,Y 323.525,Z 1203.699,A -85,B 0,C 180,E1 16565.664,E2 16565.664} C_VEL
LIN {X 0,Y 325.185,Z 1204.475,A -85,B 0,C 180,E1 16562.467,E2 16562.467} C_VEL
LIN {X 0,Y 327.788,Z 1203.211,A -85,B 0,C 180,E1 16559.126,E2 16559.126} C_VEL
LIN {X 0,Y 330.92,Z 1200.338,A -85,B 0,C 180,E1 16556.188,E2 16556.188} C_VEL
LIN {X 0,Y 335.109,Z 1195.426,A -85,B 0,C 180,E1 16553.145,E2 16553.145} C_VEL
LIN {X 0,Y 340.201,Z 1188.487,A -85,B 0,C 180,E1 16550.185,E2 16550.185} C_VEL
LIN {X 0,Y 345.444,Z 1180.363,A -85,B 0,C 180,E1 16547.632,E2 16547.632} C_VEL
LIN {X 0,Y 351.034,Z 1171.003,A -85,B 0,C 180,E1 16545.315,E2 16545.315} C_VEL
LIN {X 0,Y 357.647,Z 1158.7,A -85,B 0,C 180,E1 16542.929,E2 16542.929} C_VEL
LIN {X 0,Y 364.514,Z 1144.481,A -85,B 0,C 180,E1 16540.782,E2 16540.782} C_VEL
LIN {X 0,Y 370.752,Z 1130.072,A -85,B 0,C 180,E1 16539.063,E2 16539.063} C_VEL
LIN {X 0,Y 376.925,Z 1114.094,A -85,B 0,C 180,E1 16537.542,E2 16537.542} C_VEL
LIN {X 0,Y 383.935,Z 1093.541,A -85,B 0,C 180,E1 16536.029,E2 16536.029} C_VEL
LIN {X 0,Y 393.591,Z 1065.396,A -85,B 0,C 180,E1 16534.363,E2 16534.363} C_VEL
LIN {X 0,Y 403.702,Z 1034.329,A -85,B 0,C 180,E1 16532.888,E2 16532.888} C_VEL
LIN {X 0,Y 412.928,Z 1001.674,A -85,B 0,C 180,E1 16531.587,E2 16531.587} C_VEL
LIN {X 0,Y 419.329,Z 974.472,A -85,B 0,C 180,E1 16530.639,E2 16530.639} C_VEL
LIN {X 0,Y 421.602,Z 960.59,A -85,B 0,C 180,E1 16529.263,E2 16529.263} C_VEL
LIN {X 0,Y 432.565,Z 944.096,A -85,B 0,C 180,E1 16527.073,E2 16527.073} C_VEL
LIN {X 0,Y 423.363,Z 960.217,A -85,B 0,C 180,E1 16524.479,E2 16524.479} C_VEL
LIN {X 0,Y 418.824,Z 971.064,A -85,B 0,C 180,E1 16522.632,E2 16522.632} C_VEL
LIN {X 0,Y 418.295,Z 987.214,A -85,B 0,C 180,E1 16520.223,E2 16520.223} C_VEL
LIN {X 0,Y 414.835,Z 1003.362,A -85,B 0,C 180,E1 16519.928,E2 16519.928} C_VEL
LIN {X 0,Y 408.812,Z 1027.822,A -85,B 0,C 180,E1 16519.464,E2 16519.464} C_VEL
LIN {X 0,Y 403.2,Z 1048.068,A -85,B 0,C 180,E1 16518.816,E2 16518.816} C_VEL
LIN {X 0,Y 395.384,Z 1073.675,A -85,B 0,C 180,E1 16517.702,E2 16517.702} C_VEL
LIN {X 0,Y 386.619,Z 1098.961,A -85,B 0,C 180,E1 16516.287,E2 16516.287} C_VEL
LIN {X 0,Y 378.034,Z 1121.779,A -85,B 0,C 180,E1 16514.643,E2 16514.643} C_VEL
LIN {X 0,Y 369.379,Z 1143.62,A -85,B 0,C 180,E1 16512.691,E2 16512.691} C_VEL
LIN {X 0,Y 360.773,Z 1163.99,A -85,B 0,C 180,E1 16510.428,E2 16510.428} C_VEL
LIN {X 0,Y 352.343,Z 1183.085,A -85,B 0,C 180,E1 16507.801,E2 16507.801} C_VEL
LIN {X 0,Y 344.552,Z 1200.473,A -85,B 0,C 180,E1 16504.865,E2 16504.865} C_VEL
LIN {X 0,Y 337.911,Z 1215.505,A -85,B 0,C 180,E1 16501.78,E2 16501.78} C_VEL
LIN {X 0,Y 331.883,Z 1229.718,A -85,B 0,C 180,E1 16498.226,E2 16498.226} C_VEL
LIN {X 0,Y 327.258,Z 1241.692,A -85,B 0,C 180,E1 16494.55,E2 16494.55} C_VEL
LIN {X 0,Y 324.097,Z 1251.198,A -85,B 0,C 180,E1 16490.967,E2 16490.967} C_VEL
LIN {X 0,Y 322.046,Z 1259.644,A -85,B 0,C 180,E1 16487.152,E2 16487.152} C_VEL
LIN {X 0,Y 320.947,Z 1269.649,A -85,B 0,C 180,E1 16483.51,E2 16483.51} C_VEL
LIN {X 0,Y 320.49,Z 1277.26,A -85,B 0,C 180,E1 16480.059,E2 16480.059} C_VEL
LIN {X 0,Y 320.443,Z 1282.674,A -85,B 0,C 180,E1 16476.807,E2 16476.807} C_VEL
LIN {X 0,Y 320.508,Z 1286.844,A -85,B 0,C 180,E1 16473.396,E2 16473.396} C_VEL
LIN {X 0,Y 320.52,Z 1289.132,A -85,B 0,C 180,E1 16470.355,E2 16470.355} C_VEL
LIN {X 0,Y 320.356,Z 1290.308,A -85,B 0,C 180,E1 16467.135,E2 16467.135} C_VEL
LIN {X 0,Y 320.168,Z 1289.98,A -85,B 0,C 180,E1 16463.722,E2 16463.722} C_VEL
LIN {X 0,Y 320.268,Z 1288.253,A -85,B 0,C 180,E1 16460.11,E2 16460.11} C_VEL
LIN {X 0,Y 321.115,Z 1284.52,A -85,B 0,C 180,E1 16456.125,E2 16456.125} C_VEL
LIN {X 0,Y 323.128,Z 1278.776,A -85,B 0,C 180,E1 16451.972,E2 16451.972} C_VEL
LIN {X 0,Y 326.372,Z 1271.555,A -85,B 0,C 180,E1 16448.05,E2 16448.05} C_VEL
LIN {X 0,Y 331.266,Z 1262.085,A -85,B 0,C 180,E1 16444.043,E2 16444.043} C_VEL
LIN {X 0,Y 337.781,Z 1250.634,A -85,B 0,C 180,E1 16440.176,E2 16440.176} C_VEL
LIN {X 0,Y 345.999,Z 1237.278,A -85,B 0,C 180,E1 16436.496,E2 16436.496} C_VEL
LIN {X 0,Y 356.418,Z 1221.273,A -85,B 0,C 180,E1 16432.902,E2 16432.902} C_VEL
LIN {X 0,Y 368.775,Z 1203.163,A -85,B 0,C 180,E1 16429.606,E2 16429.606} C_VEL
LIN {X 0,Y 381.849,Z 1184.746,A -85,B 0,C 180,E1 16426.885,E2 16426.885} C_VEL
LIN {X 0,Y 395.937,Z 1165.474,A -85,B 0,C 180,E1 16424.588,E2 16424.588} C_VEL
LIN {X 0,Y 399.856,Z 1160.05,A -85,B 0,C 180,E1 16424.019,E2 16424.019} C_VEL
LIN {X 0,Y 385.72,Z 1178.223,A -85,B 0,C 180,E1 16421.577,E2 16421.577} C_VEL
LIN {X 0,Y 372.493,Z 1195.234,A -85,B 0,C 180,E1 16418.715,E2 16418.715} C_VEL
LIN {X 0,Y 360.895,Z 1210.258,A -85,B 0,C 180,E1 16415.579,E2 16415.579} C_VEL
LIN {X 0,Y 350.475,Z 1223.856,A -85,B 0,C 180,E1 16412.05,E2 16412.05} C_VEL
LIN {X 0,Y 341.731,Z 1235.353,A -85,B 0,C 180,E1 16408.295,E2 16408.295} C_VEL
LIN {X 0,Y 334.898,Z 1244.459,A -85,B 0,C 180,E1 16404.52,E2 16404.52} C_VEL
LIN {X 0,Y 329.751,Z 1251.481,A -85,B 0,C 180,E1 16400.78,E2 16400.78} C_VEL
LIN {X 0,Y 325.612,Z 1257.129,A -85,B 0,C 180,E1 16396.641,E2 16396.641} C_VEL
LIN {X 0,Y 322.973,Z 1260.634,A -85,B 0,C 180,E1 16392.698,E2 16392.698} C_VEL
LIN {X 0,Y 321.333,Z 1262.531,A -85,B 0,C 180,E1 16388.59,E2 16388.59} C_VEL
LIN {X 0,Y 320.566,Z 1262.712,A -85,B 0,C 180,E1 16384.831,E2 16384.831} C_VEL
LIN {X 0,Y 320.257,Z 1261.335,A -85,B 0,C 180,E1 16381.252,E2 16381.252} C_VEL
LIN {X 0,Y 320.162,Z 1258.508,A -85,B 0,C 180,E1 16377.673,E2 16377.673} C_VEL
LIN {X 0,Y 320.245,Z 1254.407,A -85,B 0,C 180,E1 16374.266,E2 16374.266} C_VEL
LIN {X 0,Y 320.58,Z 1248.71,A -85,B 0,C 180,E1 16370.847,E2 16370.847} C_VEL
LIN {X 0,Y 321.354,Z 1241.013,A -85,B 0,C 180,E1 16367.237,E2 16367.237} C_VEL
LIN {X 0,Y 322.642,Z 1231.887,A -85,B 0,C 180,E1 16363.804,E2 16363.804} C_VEL
LIN {X 0,Y 324.581,Z 1220.693,A -85,B 0,C 180,E1 16360.38,E2 16360.38} C_VEL
LIN {X 0,Y 327.092,Z 1208.051,A -85,B 0,C 180,E1 16357.156,E2 16357.156} C_VEL
LIN {X 0,Y 330.302,Z 1193.107,A -85,B 0,C 180,E1 16353.963,E2 16353.963} C_VEL
LIN {X 0,Y 333.782,Z 1177.558,A -85,B 0,C 180,E1 16351.164,E2 16351.164} C_VEL
LIN {X 0,Y 337.667,Z 1160.2,A -85,B 0,C 180,E1 16348.522,E2 16348.522} C_VEL
LIN {X 0,Y 341.901,Z 1140.681,A -85,B 0,C 180,E1 16346.042,E2 16346.042} C_VEL
LIN {X 0,Y 346.079,Z 1120.293,A -85,B 0,C 180,E1 16343.886,E2 16343.886} C_VEL
LIN {X 0,Y 349.935,Z 1099.962,A -85,B 0,C 180,E1 16342.096,E2 16342.096} C_VEL
LIN {X 0,Y 353.689,Z 1077.96,A -85,B 0,C 180,E1 16340.499,E2 16340.499} C_VEL
LIN {X 0,Y 357.153,Z 1054.697,A -85,B 0,C 180,E1 16339.146,E2 16339.146} C_VEL
LIN {X 0,Y 360.054,Z 1031.279,A -85,B 0,C 180,E1 16338.084,E2 16338.084} C_VEL
LIN {X 0,Y 362.436,Z 1006.863,A -85,B 0,C 180,E1 16337.267,E2 16337.267} C_VEL
LIN {X 0,Y 380.292,Z 800.407,A -85,B 0,C 180,E1 16331.832,E2 16331.832} C_VEL
LIN {X 0,Y 366.037,Z 772.253,A -85,B 0,C 180,E1 16329.127,E2 16329.127} C_VEL
LIN {X 0,Y 352.098,Z 746.519,A -85,B 0,C 180,E1 16326.283,E2 16326.283} C_VEL
LIN {X 0,Y 338.392,Z 722.966,A -85,B 0,C 180,E1 16323.266,E2 16323.266} C_VEL
LIN {X 0,Y 332.77,Z 713.611,A -85,B 0,C 180,E1 16321.929,E2 16321.929} C_VEL
LIN {X 0,Y 326.754,Z 700.309,A -85,B 0,C 180,E1 16318.916,E2 16318.916} C_VEL
LIN {X 0,Y 324.336,Z 695.495,A -85,B 0,C 180,E1 16317.746,E2 16317.746} C_VEL
LIN {X 0,Y 323.278,Z 692.402,A -85,B 0,C 180,E1 16317.028,E2 16317.028} C_VEL
LIN {X 0,Y 323.274,Z 692.402,A -85,B 0,C 180,E1 16312.555,E2 16312.555} C_VEL
LIN {X 0,Y 323.281,Z 692.401,A -85,B 0,C 180,E1 16308.205,E2 16308.205} C_VEL
LIN {X 0,Y 323.271,Z 692.383,A -85,B 0,C 180,E1 16303.779,E2 16303.779} C_VEL
LIN {X 0,Y 323.269,Z 692.385,A -85,B 0,C 180,E1 16299.358,E2 16299.358} C_VEL
LIN {X 0,Y 323.269,Z 692.388,A -85,B 0,C 180,E1 16294.971,E2 16294.971} C_VEL
LIN {X 0,Y 323.28,Z 692.385,A -85,B 0,C 180,E1 16290.534,E2 16290.534} C_VEL
LIN {X 0,Y 323.27,Z 692.385,A -85,B 0,C 180,E1 16286.101,E2 16286.101} C_VEL
LIN {X 0,Y 323.272,Z 692.386,A -85,B 0,C 180,E1 16281.799,E2 16281.799} C_VEL
LIN {X 0,Y 323.3,Z 692.628,A -85,B 0,C 180,E1 16279.309,E2 16279.309} C_VEL
LIN {X 0,Y 324.789,Z 696.168,A -85,B 0,C 180,E1 16278.099,E2 16278.099} C_VEL
LIN {X 0,Y 325.691,Z 697.324,A -85,B 0,C 180,E1 16277.593,E2 16277.593} C_VEL
LIN {X 0,Y 327.271,Z 700.916,A -85,B 0,C 180,E1 16276.396,E2 16276.396} C_VEL
LIN {X 0,Y 328.51,Z 703.447,A -85,B 0,C 180,E1 16275.55,E2 16275.55} C_VEL
LIN {X 0,Y 330.56,Z 707.454,A -85,B 0,C 180,E1 16274.205,E2 16274.205} C_VEL
LIN {X 0,Y 334.714,Z 716.056,A -85,B 0,C 180,E1 16271.542,E2 16271.542} C_VEL
LIN {X 0,Y 340.051,Z 727.645,A -85,B 0,C 180,E1 16268.257,E2 16268.257} C_VEL
LIN {X 0,Y 346.078,Z 741.61,A -85,B 0,C 180,E1 16264.687,E2 16264.687} C_VEL
LIN {X 0,Y 352.196,Z 757.024,A -85,B 0,C 180,E1 16261.146,E2 16261.146} C_VEL
LIN {X 0,Y 358.36,Z 774.067,A -85,B 0,C 180,E1 16257.611,E2 16257.611} C_VEL
LIN {X 0,Y 364.221,Z 792.092,A -85,B 0,C 180,E1 16254.218,E2 16254.218} C_VEL
LIN {X 0,Y 366.905,Z 801.147,A -85,B 0,C 180,E1 16252.628,E2 16252.628} C_VEL
LIN {X 0,Y 358.429,Z 844.037,A -85,B 0,C 180,E1 16247.906,E2 16247.906} C_VEL
LIN {X 0,Y 350.64,Z 887.76,A -85,B 0,C 180,E1 16243.076,E2 16243.076} C_VEL
LIN {X 0,Y 345.01,Z 924.125,A -85,B 0,C 180,E1 16239.09,E2 16239.09} C_VEL
LIN {X 0,Y 345.247,Z 936.299,A -85,B 0,C 180,E1 16238.584,E2 16238.584} C_VEL
LIN {X 0,Y 339.365,Z 1006.715,A -85,B 0,C 180,E1 16236.021,E2 16236.021} C_VEL
LIN {X 0,Y 338.128,Z 1021.601,A -85,B 0,C 180,E1 16235.428,E2 16235.428} C_VEL
LIN {X 0,Y 336.555,Z 1029.067,A -85,B 0,C 180,E1 16235.181,E2 16235.181} C_VEL
LIN {X 0,Y 329.083,Z 1048.722,A -85,B 0,C 180,E1 16234.678,E2 16234.678} C_VEL
LIN {X 0,Y 327.912,Z 1055.103,A -85,B 0,C 180,E1 16234.422,E2 16234.422} C_VEL
LIN {X 0,Y 326.162,Z 1081.84,A -85,B 0,C 180,E1 16233.071,E2 16233.071} C_VEL
LIN {X 0,Y 324.701,Z 1098.854,A -85,B 0,C 180,E1 16231.879,E2 16231.879} C_VEL
LIN {X 0,Y 322.892,Z 1115.944,A -85,B 0,C 180,E1 16230.315,E2 16230.315} C_VEL
LIN {X 0,Y 320.937,Z 1132.499,A -85,B 0,C 180,E1 16228.367,E2 16228.367} C_VEL
LIN {X 0,Y 319.205,Z 1146.05,A -85,B 0,C 180,E1 16226.386,E2 16226.386} C_VEL
LIN {X 0,Y 317.527,Z 1159.075,A -85,B 0,C 180,E1 16224.056,E2 16224.056} C_VEL
LIN {X 0,Y 316.102,Z 1170.466,A -85,B 0,C 180,E1 16221.527,E2 16221.527} C_VEL
LIN {X 0,Y 315.072,Z 1180.174,A -85,B 0,C 180,E1 16218.887,E2 16218.887} C_VEL
LIN {X 0,Y 314.38,Z 1188.913,A -85,B 0,C 180,E1 16215.874,E2 16215.874} C_VEL
LIN {X 0,Y 314.171,Z 1195.618,A -85,B 0,C 180,E1 16212.873,E2 16212.873} C_VEL
LIN {X 0,Y 314.464,Z 1200.967,A -85,B 0,C 180,E1 16209.517,E2 16209.517} C_VEL
LIN {X 0,Y 315.356,Z 1204.222,A -85,B 0,C 180,E1 16206.189,E2 16206.189} C_VEL
LIN {X 0,Y 316.84,Z 1205.563,A -85,B 0,C 180,E1 16203.075,E2 16203.075} C_VEL
LIN {X 0,Y 319.353,Z 1205.061,A -85,B 0,C 180,E1 16199.641,E2 16199.641} C_VEL
LIN {X 0,Y 322.622,Z 1202.663,A -85,B 0,C 180,E1 16196.446,E2 16196.446} C_VEL
LIN {X 0,Y 326.818,Z 1198.433,A -85,B 0,C 180,E1 16193.324,E2 16193.324} C_VEL
LIN {X 0,Y 331.943,Z 1192.223,A -85,B 0,C 180,E1 16190.289,E2 16190.289} C_VEL
LIN {X 0,Y 337.971,Z 1183.854,A -85,B 0,C 180,E1 16187.354,E2 16187.354} C_VEL
LIN {X 0,Y 344.507,Z 1173.715,A -85,B 0,C 180,E1 16184.685,E2 16184.685} C_VEL
LIN {X 0,Y 350.929,Z 1162.669,A -85,B 0,C 180,E1 16182.421,E2 16182.421} C_VEL
LIN {X 0,Y 357.528,Z 1150.27,A -85,B 0,C 180,E1 16180.391,E2 16180.391} C_VEL
LIN {X 0,Y 364.464,Z 1135.844,A -85,B 0,C 180,E1 16178.515,E2 16178.515} C_VEL
LIN {X 0,Y 371.376,Z 1119.588,A -85,B 0,C 180,E1 16176.853,E2 16176.853} C_VEL
LIN {X 0,Y 377.618,Z 1102.979,A -85,B 0,C 180,E1 16175.519,E2 16175.519} C_VEL
LIN {X 0,Y 387.378,Z 1076.339,A -85,B 0,C 180,E1 16173.808,E2 16173.808} C_VEL
LIN {X 0,Y 397.883,Z 1046.559,A -85,B 0,C 180,E1 16172.295,E2 16172.295} C_VEL
LIN {X 0,Y 407.418,Z 1015.973,A -85,B 0,C 180,E1 16171.007,E2 16171.007} C_VEL
LIN {X 0,Y 415.276,Z 986.246,A -85,B 0,C 180,E1 16169.946,E2 16169.946} C_VEL
LIN {X 0,Y 417.321,Z 977.335,A -85,B 0,C 180,E1 16169.632,E2 16169.632} C_VEL
LIN {X 0,Y 420.201,Z 962.385,A -85,B 0,C 180,E1 16168.112,E2 16168.112} C_VEL
LIN {X 0,Y 425.895,Z 954.012,A -85,B 0,C 180,E1 16166.997,E2 16166.997} C_VEL
LIN {X 0,Y 418.107,Z 968.094,A -85,B 0,C 180,E1 16164.661,E2 16164.661} C_VEL
LIN {X 0,Y 415.907,Z 986.797,A -85,B 0,C 180,E1 16161.823,E2 16161.823} C_VEL
LIN {X 0,Y 415.681,Z 991.028,A -85,B 0,C 180,E1 16161.212,E2 16161.212} C_VEL
LIN {X 0,Y 408.354,Z 1021.343,A -85,B 0,C 180,E1 16160.695,E2 16160.695} C_VEL
LIN {X 0,Y 402.509,Z 1041.931,A -85,B 0,C 180,E1 16160.135,E2 16160.135} C_VEL
LIN {X 0,Y 394.719,Z 1066.931,A -85,B 0,C 180,E1 16159.122,E2 16159.122} C_VEL
LIN {X 0,Y 386.227,Z 1091.014,A -85,B 0,C 180,E1 16157.873,E2 16157.873} C_VEL
LIN {X 0,Y 377.603,Z 1113.37,A -85,B 0,C 180,E1 16156.4,E2 16156.4} C_VEL
LIN {X 0,Y 368.703,Z 1135.017,A -85,B 0,C 180,E1 16154.615,E2 16154.615} C_VEL
LIN {X 0,Y 359.379,Z 1156.315,A -85,B 0,C 180,E1 16152.427,E2 16152.427} C_VEL
LIN {X 0,Y 350.552,Z 1175.342,A -85,B 0,C 180,E1 16149.984,E2 16149.984} C_VEL
LIN {X 0,Y 342.615,Z 1191.984,A -85,B 0,C 180,E1 16147.371,E2 16147.371} C_VEL
LIN {X 0,Y 334.588,Z 1208.644,A -85,B 0,C 180,E1 16144.178,E2 16144.178} C_VEL
LIN {X 0,Y 327.582,Z 1223.614,A -85,B 0,C 180,E1 16140.643,E2 16140.643} C_VEL
LIN {X 0,Y 321.977,Z 1236.299,A -85,B 0,C 180,E1 16136.959,E2 16136.959} C_VEL
LIN {X 0,Y 317.945,Z 1246.507,A -85,B 0,C 180,E1 16133.321,E2 16133.321} C_VEL
LIN {X 0,Y 315.108,Z 1255.26,A -85,B 0,C 180,E1 16129.459,E2 16129.459} C_VEL
LIN {X 0,Y 313.916,Z 1260.282,A -85,B 0,C 180,E1 16126.846,E2 16126.846} C_VEL
LIN {X 0,Y 312.922,Z 1269.618,A -85,B 0,C 180,E1 16123.298,E2 16123.298} C_VEL
LIN {X 0,Y 312.502,Z 1277.103,A -85,B 0,C 180,E1 16119.772,E2 16119.772} C_VEL
LIN {X 0,Y 312.472,Z 1282.477,A -85,B 0,C 180,E1 16116.428,E2 16116.428} C_VEL
LIN {X 0,Y 312.554,Z 1286.531,A -85,B 0,C 180,E1 16112.931,E2 16112.931} C_VEL
LIN {X 0,Y 312.534,Z 1288.749,A -85,B 0,C 180,E1 16109.814,E2 16109.814} C_VEL
LIN {X 0,Y 312.315,Z 1289.836,A -85,B 0,C 180,E1 16106.326,E2 16106.326} C_VEL
LIN {X 0,Y 312.167,Z 1289.379,A -85,B 0,C 180,E1 16102.822,E2 16102.822} C_VEL
LIN {X 0,Y 312.445,Z 1287.199,A -85,B 0,C 180,E1 16098.74,E2 16098.74} C_VEL
LIN {X 0,Y 313.664,Z 1283.293,A -85,B 0,C 180,E1 16094.655,E2 16094.655} C_VEL
LIN {X 0,Y 316.183,Z 1277.36,A -85,B 0,C 180,E1 16090.458,E2 16090.458} C_VEL
LIN {X 0,Y 320.45,Z 1269.145,A -85,B 0,C 180,E1 16086.099,E2 16086.099} C_VEL
LIN {X 0,Y 326.537,Z 1258.871,A -85,B 0,C 180,E1 16081.862,E2 16081.862} C_VEL
LIN {X 0,Y 334.102,Z 1247.222,A -85,B 0,C 180,E1 16078.011,E2 16078.011} C_VEL
LIN {X 0,Y 343.876,Z 1233.058,A -85,B 0,C 180,E1 16074.219,E2 16074.219} C_VEL
